// SIMATIC S7-200 SMART project (STEP 7-Micro/WIN SMART), CPU ST60

SYMBOL_TABLE V区符号
参数传输成功           V0.0     // 接收工控机传来的数据传输成功信号
参数是否更新           V0.1
挡板自动控制完成标志       V0.2
挡板电机开关           V0.3
挡板手动向内           V0.4
挡板手动向外           V0.5
挡板一键调节           V0.6
下料电机开关           V0.7
下料手动向前           V1.0
下料手动向后           V1.1
冷却电机开关           V1.2
冷却电机点动向内         V1.3
冷却电机点动向外         V1.4
冷柜一键调节           V1.5
调试按钮             V1.6
恢复出厂设置           V1.7
报警信息1用           VB2
V型架未处于停止位        V3.0     // 用于显示屏显示报警信息
系统处于急停模式         V3.1     // 用于显示屏显示报警信息
挡板运动超过左限制区       V3.2     // 用于显示屏显示报警信息
挡板运动超过右限制区       V3.3     // 用于显示屏显示报警信息
下料小车运动超过前限制      V3.4     // 用于显示屏显示报警信息
下料小车运动超过后限制      V3.5     // 用于显示屏显示报警信息
冷却风柜运动超过左限制      V3.6     // 用于显示屏显示报警信息
冷却风柜运动超过右限制      V3.7     // 用于显示屏显示报警信息
报警信息2用           VB4
上料步进故障           V5.0
上料传动故障           V5.1
上料夹料位报警          V5.2
请先建立绝对坐标         V5.3
链传动限位传感器报警       V5.4
挡板参数改变请初始化       V5.5
冷却参数改变请初始化       V5.6
报警灯红灯常开          V8.0
报警灯黄灯常开          V8.1
报警灯绿灯常开          V8.2
报警灯红灯闪烁和蜂鸣       V8.4
报警灯黄灯闪烁          V8.5
报警灯绿灯闪烁          V8.6
挡板电机手动运行         V10.0
冷却电机手动运行         V10.1
下料电机手动运行         V10.2
挡板手动一键调节         V10.3
挡板一键调节完成标志       V10.4
冷却手动一键调节         V10.5
冷却一键调节完成标志       V10.6
挡板点动向外           V11.1
挡板点动向内           V11.2
挡板电机查找原点按钮       V11.3
下料电机查找原点按钮       V11.4
冷却电机查找原点按钮       V11.5
挡板自动控制           V11.6
下料下移一个工位         V11.7
下料启动按钮           V12.0
下料手动完成标志         V12.1
下料手动回到原点         V12.2
下料手动回到底部         V12.3
冷却自动控制           V12.4
挡板电机查找原点         V12.5
下料电机查找原点         V12.6
冷却电机查找原点         V12.7
冷却点动向内           V13.0
冷却点动向外           V13.1
下料点动向前           V13.2
下料点动向后           V13.3
冷却启动按钮           V13.4
放料完成开关           V13.5    // 不再需要上杆件后，按下此按键，上料架上杆件自动向前
上料步进停止位          V13.6
上料杆件序号确认         V13.7
挡板电机CTRL错误参数     VB16
挡板电机RSEEK错误参数    VB18
挡板电机函数完成标志位      V20.1
挡板电机当前运动方向       V20.2
挡板电机查找原点完成位      V20.3    // 查找到原点动作已完成
挡板电机GOTO完成位      V20.4
挡板电机GOTO错误参数     VB21
挡板电机当前位置         VD24
挡板电机当前速度         VD28
上一次挡板停止位置        VD32
挡板电机移动位置         VD44
挡板电机速度           VD48
挡板电机移动模式         VB41
挡板电机停止运动轴        V40.1
挡板电机运动方向         V40.2
挡板当前实际位置         VD52
挡板相对运动距离         VD56
冷却电机初始化完成位       V60.1
冷却电机当前运动方向       V60.2
冷却电机查找原点完成位      V60.3
冷却电机GOTO完成位      V60.4
冷却电机GOTO错误参数     VB61
冷却电机当前位置         VD64
冷却电机当前速度         VD68
冷柜电机CTRL错误参数     VB72
冷柜电机RSEEK错误参数    VB75
冷却电机移动位置         VD84
冷却电机速度           VD88
冷却电机移动模式         VB81
冷却电机停止运动轴        V80.1
冷却电机运动方向         V80.2
下料电机函数完成标志位      V100.1
下料电机当前运动方向       V100.2
下料电机查找原点完成位      V100.3
下料电机GOTO完成位      V100.4
下料电机错误参数         VB101
下料电机当前位置         VD104
下料电机当前速度         VD108
下料电机当前位置上限       VD112
下料电机当前位置下限       VD116
下料电机移动位置         VD124
下料电机速度           VD128
下料电机移动模式         VB121
下料电机停止运动轴        V120.1
下料电机运动方向         V120.2
杆件编号             VB136
上一杆件数据           VD140
当前杆件数据           VD144
下料电机运动到杆件放置      VD150
下料电机下移一个杆件位      VD154
下料电机二号杆件位置       VD158
下料电机三号杆件位置       VD162
下料电机四号杆件位置       VD166
下料电机五号杆件位置       VD170
小车下料终点位置         VD174
挡板长度             VD180    // 定位零点以后，挡板能调节的最大长度
挡板预留长度           VD184    // 根据杆件的长度加上预留长度为实际调节距离
挡板临时变量           VD188    // 挡板长度减去当前杆件长度
挡板预留长度临时变量       VD192
轴0运动组态用          VB200    // VB200-VB292为轴0占用
轴1运动组态用          VB293    // VB293-VB385为轴1占用
轴2运动组态用          VB386    // VB386-VB478为轴2占用
链传动使能按钮          V480.0
链传动低速按钮          V480.1
链传动高速按钮          V480.2
链传动一个工位按钮        V480.3   // 链传动机构运动一个杆位按钮
链传动自动运行          V480.4
杆件编号1            V500.0   // VB500-VB748存放杆件编号和长度
杆件编号2            V500.1   // VB500-VB748存放杆件编号和长度
杆件编号3            V500.2   // VB500-VB748存放杆件编号和长度
杆件编号4            V500.3   // VB500-VB748存放杆件编号和长度
杆件编号5            V500.4   // VB500-VB748存放杆件编号和长度
杆件编号6            V500.5   // VB500-VB748存放杆件编号和长度
杆件编号7            V500.6   // VB500-VB748存放杆件编号和长度
杆件编号8            V500.7   // VB500-VB748存放杆件编号和长度
杆件编号9            V501.0   // VB500-VB748存放杆件编号和长度
杆件编号10           V501.1   // VB500-VB748存放杆件编号和长度
杆件编号11           V501.2   // VB500-VB748存放杆件编号和长度
杆件编号12           V501.3   // VB500-VB748存放杆件编号和长度
杆件编号13           V501.4   // VB500-VB748存放杆件编号和长度
杆件编号14           V501.5   // VB500-VB748存放杆件编号和长度
杆件编号15           V501.6   // VB500-VB748存放杆件编号和长度
杆件编号16           V501.7   // VB500-VB748存放杆件编号和长度
杆件编号17           V502.0   // VB500-VB748存放杆件编号和长度
杆件编号18           V502.1   // VB500-VB748存放杆件编号和长度
杆件编号19           V502.2   // VB500-VB748存放杆件编号和长度
杆件编号20           V502.3   // VB500-VB748存放杆件编号和长度
杆件编号21           V502.4   // VB500-VB748存放杆件编号和长度
杆件编号22           V502.5   // VB500-VB748存放杆件编号和长度
杆件编号23           V502.6   // VB500-VB748存放杆件编号和长度
杆件编号24           V502.7   // VB500-VB748存放杆件编号和长度
杆件编号25           V503.0   // VB500-VB748存放杆件编号和长度
杆件编号26           V503.1   // VB500-VB748存放杆件编号和长度
杆件编号27           V503.2   // VB500-VB748存放杆件编号和长度
杆件编号28           V503.3   // VB500-VB748存放杆件编号和长度
杆件编号29           V503.4   // VB500-VB748存放杆件编号和长度
杆件编号30           V503.5   // VB500-VB748存放杆件编号和长度
杆件编号31           V503.6   // VB500-VB748存放杆件编号和长度
杆件编号32           V503.7   // VB500-VB748存放杆件编号和长度
杆件编号33           V504.0   // VB500-VB748存放杆件编号和长度
杆件编号34           V504.1   // VB500-VB748存放杆件编号和长度
杆件编号35           V504.2   // VB500-VB748存放杆件编号和长度
杆件编号36           V504.3   // VB500-VB748存放杆件编号和长度
杆件编号37           V504.4   // VB500-VB748存放杆件编号和长度
杆件编号38           V504.5   // VB500-VB748存放杆件编号和长度
杆件编号39           V504.6   // VB500-VB748存放杆件编号和长度
杆件编号40           V504.7   // VB500-VB748存放杆件编号和长度
杆件编号41           V505.0   // VB500-VB748存放杆件编号和长度
杆件编号42           V505.1   // VB500-VB748存放杆件编号和长度
杆件编号43           V505.2   // VB500-VB748存放杆件编号和长度
杆件编号44           V505.3   // VB500-VB748存放杆件编号和长度
杆件编号45           V505.4   // VB500-VB748存放杆件编号和长度
杆件编号46           V505.5   // VB500-VB748存放杆件编号和长度
杆件编号47           V505.6   // VB500-VB748存放杆件编号和长度
杆件编号48           V505.7   // VB500-VB748存放杆件编号和长度
杆件编号49           V506.0   // VB500-VB748存放杆件编号和长度
杆件编号50           V506.1   // VB500-VB748存放杆件编号和长度
杆件编号临时变量         VB510
杆件编号标志位1         V520.1
杆件编号标志位2         V520.2
杆件编号标志位3         V520.3
杆件编号标志位4         V520.4
杆件编号标志位5         V520.5
杆件编号标志位6         V520.6
杆件编号标志位7         V520.7
杆件编号标志位8         V521.0
杆件编号标志位9         V521.1
杆件编号标志位10        V521.2
杆件编号标志位11        V521.3
杆件编号标志位12        V521.4
杆件编号标志位13        V521.5
杆件编号标志位14        V521.6
杆件编号标志位15        V521.7
杆件编号标志位16        V522.0
杆件编号标志位17        V522.1
杆件编号标志位18        V522.2
杆件编号标志位19        V522.3
杆件编号标志位20        V522.4
杆件编号标志位21        V522.5
杆件编号标志位22        V522.6
杆件编号标志位23        V522.7
杆件编号标志位24        V523.0
杆件编号标志位25        V523.1
杆件编号标志位26        V523.2
杆件编号标志位27        V523.3
杆件编号标志位28        V523.4
杆件编号标志位29        V523.5
杆件编号标志位30        V523.6
杆件编号标志位31        V523.7
杆件编号标志位32        V524.0
杆件编号标志位33        V524.1
杆件编号标志位34        V524.2
杆件编号标志位35        V524.3
杆件编号标志位36        V524.4
杆件编号标志位37        V524.5
杆件编号标志位38        V524.6
杆件编号标志位39        V524.7
杆件编号标志位40        V525.0
杆件编号标志位41        V525.1
杆件编号标志位42        V525.2
杆件编号标志位43        V525.3
杆件编号标志位44        V525.4
杆件编号标志位45        V525.5
杆件编号标志位46        V525.6
杆件编号标志位47        V525.7
杆件编号标志位48        V526.0
杆件编号标志位49        V526.1
杆件编号标志位50        V526.2
上料架位置1           VB540
上料架位置2           VB541
上料架位置3           VB542
上料架位置4           VB543
上料架位置5           VB544
上料架位置6           VB545
上料架位置7           VB546
上料架位置8           VB547
上料架位置9           VB548
上料架位置10          VB549
上料架位置11          VB550
上料架位置12          VB551
上料架位置13          VB552
上料架位置14          VB553
上料架位置15          VB554
上料架位置16          VB555
上料架位置17          VB556
上料架位置18          VB557
上料架位置19          VB558
上料架位置20          VB559
上料架位置21          VB560
上料架位置22          VB561
上料架位置23          VB562
上料架位置24          VB563
上料架位置25          VB564
上料架位置26          VB565
上料架位置27          VB566
上料架位置28          VB567
上料架位置29          VB568
上料架位置30          VB569
上料架位置31          VB570
上料架位置32          VB571
上料架标志位1          V580.0
上料架标志位2          V580.1
上料架标志位3          V580.2
顺序控制延时1          VW800    // T33定时变量
顺序控制延时2          VW802    // T34定时变量
挡板手动调节延时         VW804    // T104定时变量
上料故障报警定时         VW806    // T37定时变量
链传动控制定时器         VW808    // T97定时变量
挡板运动脉冲1          VW810    // T101定时变量
下料运动脉冲1          VW812    // T102定时变量
冷却运动脉冲1          VW814    // T103定时变量
上料停止位判断定时器       VW816    // T34定时变量
冷却手动调节延时         VW818    // T105定时变量
冷柜长度             VD900    // 定位零点以后，冷却风扇能移动的最大长度
冷柜预留长度           VD904    // 冷柜长度减去杆的长度
冷柜临时变量           VD908
冷柜预留长度临时变量       VD912
挡调距离             VD916
柜调长度             VD920
下料电机当前位置temp     VD924
下料运动左区间          VD928
下料运动右区间          VD932
下料电机速度高速         VD936    // 下料变速运动，速度为高速
下料电机速度低速         VD940    // 下料变速运动，速度为低速
前后两根杆件长度差        VD960
冷柜上一杆件长度         VD964
冷柜当前杆件长度         VD968
冷柜前后杆件长度差        VD972
风柜当前实际位置         VD976
上一次风柜停止位置        VD980
风柜相对移动距离         VD984
置工件就绪            V1000.0
上料位异常信号          V1001.0
下料位允许放料信号        V1018.0
下料位启动信号          V1118.1
下料位异常信号          V1019.0
上料取件完成信号         V1200.0
下料位机器人放料完成信      V1212.0
下料小车下移信号         V1212.1
手动机器人放料完成信号      V1212.2
temp上料位异常信号      V1500.0
temp下料位异常信号      V1500.1
temp冷却位异常信号      V1500.2
挡板电机手动完成标志       VB1600
冷却电机手动完成标志       VB1602
手动跳到s_6          V3000.0
C0计数器复位          V5000.0
END_SYMBOL_TABLE

SYMBOL_TABLE 系统符号
Always_On        SM0.0    // 始终接通
First_Scan_On    SM0.1    // 仅在第一个扫描周期时接通
END_SYMBOL_TABLE

SYMBOL_TABLE S区符号
扫码启动上料           S0.0
判断杆件长度是否更新       S0.1
挡板调节             S0.2
判断夹料位是否有杆件       S0.3
开启链传动            S0.4
停止链传动            S0.5
置工件就绪回到第一步       S0.6
END_SYMBOL_TABLE

SYMBOL_TABLE 定时器符号
顺序控制延时1_10ms     T33      // 短延时，保证正确读取到判断工件有无传感器的状态
上料停止位判断延时_10ms   T34
到位传感器延时_10ms     T35      // 短延时，保证正确读取到判断工件有无传感器的状态
顺序控制延时3_100ms    T36
上料故障报警定时_100ms   T37      // 设置定时，超时则报警
下料减速区脉冲_100ms    T39
上料初始化调试          T38
链传动控制定时器_10ms    T97      // 确保链传动走出当前传感器感应区，能接收到下一个传感器信号
挡板运动脉冲1_100ms    T101     // 给一个运动脉冲信号，挡板移动到杆件长度处
下料运动脉冲1_100ms    T102     // 给一个运动脉冲信号，小车移动到机器人放料处
冷却运动脉冲1_100ms    T103     // 给一个运动脉冲信号，风柜移动到杆件长度处
挡板手动调节延时_100ms   T104     // 手动调节结束后，延时一定时间，待电机当前位置稳定后再读取
冷却手动调节街延时_100m   T105     // 手动调节结束后，延时一定时间，待电机当前位置稳定后再读取
报警灯红灯高电平_100ms   T120
报警灯红灯低电平_100ms   T121
报警灯黄灯高电平_100ms   T122
报警灯黄灯低电平_100ms   T123
报警灯绿灯高电平_100ms   T124
报警灯绿灯低电平_100ms   T125
报警蜂鸣器高电平_100ms   T126
报警蜂鸣器低电平_100ms   T127
END_SYMBOL_TABLE

ORGANIZATION_BLOCK 主程序:OB1
TITLE=
BEGIN
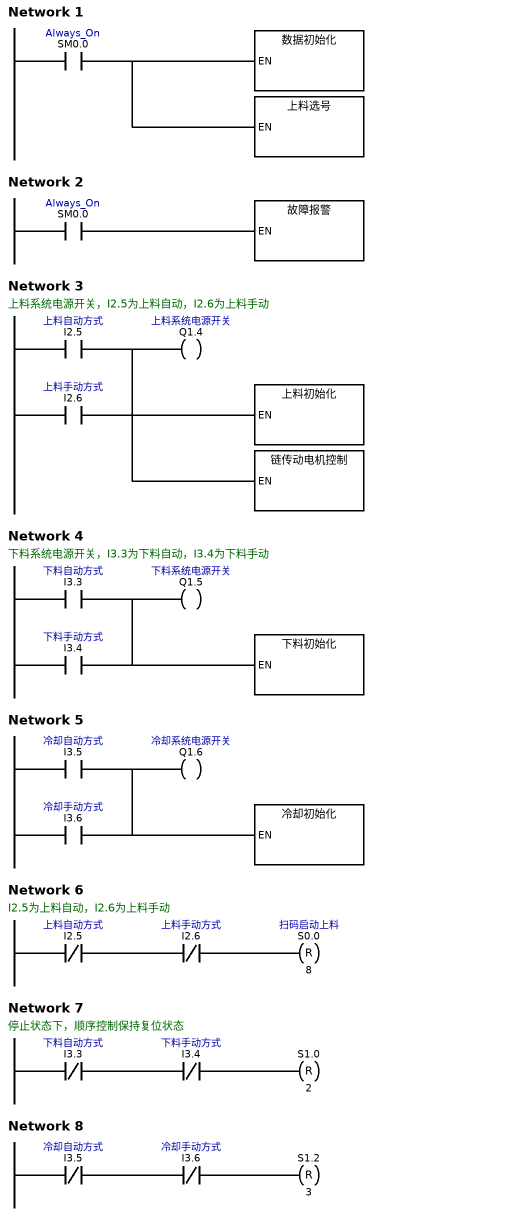
Network 1
LD     Always_On:SM0.0
CALL   数据初始化:SBR20
CALL   上料选号:SBR17
Network 2
LD     Always_On:SM0.0
CALL   故障报警:SBR21
Network 3
// 上料系统电源开关，I2.5为上料自动，I2.6为上料手动
LD     上料自动方式:I2.5
O      上料手动方式:I2.6
=      上料系统电源开关:Q1.4
CALL   上料初始化:SBR14
CALL   链传动电机控制:SBR19
Network 4
// 下料系统电源开关，I3.3为下料自动，I3.4为下料手动
LD     下料自动方式:I3.3
O      下料手动方式:I3.4
=      下料系统电源开关:Q1.5
CALL   下料初始化:SBR15
Network 5
LD     冷却自动方式:I3.5
O      冷却手动方式:I3.6
=      冷却系统电源开关:Q1.6
CALL   冷却初始化:SBR16
Network 6
// I2.5为上料自动，I2.6为上料手动
LDN    上料自动方式:I2.5
AN     上料手动方式:I2.6
R      扫码启动上料:S0.0, 8
Network 7
// 停止状态下，顺序控制保持复位状态
LDN    下料自动方式:I3.3
AN     下料手动方式:I3.4
R      S1.0, 2
Network 8
LDN    冷却自动方式:I3.5
AN     冷却手动方式:I3.6
R      S1.2, 3
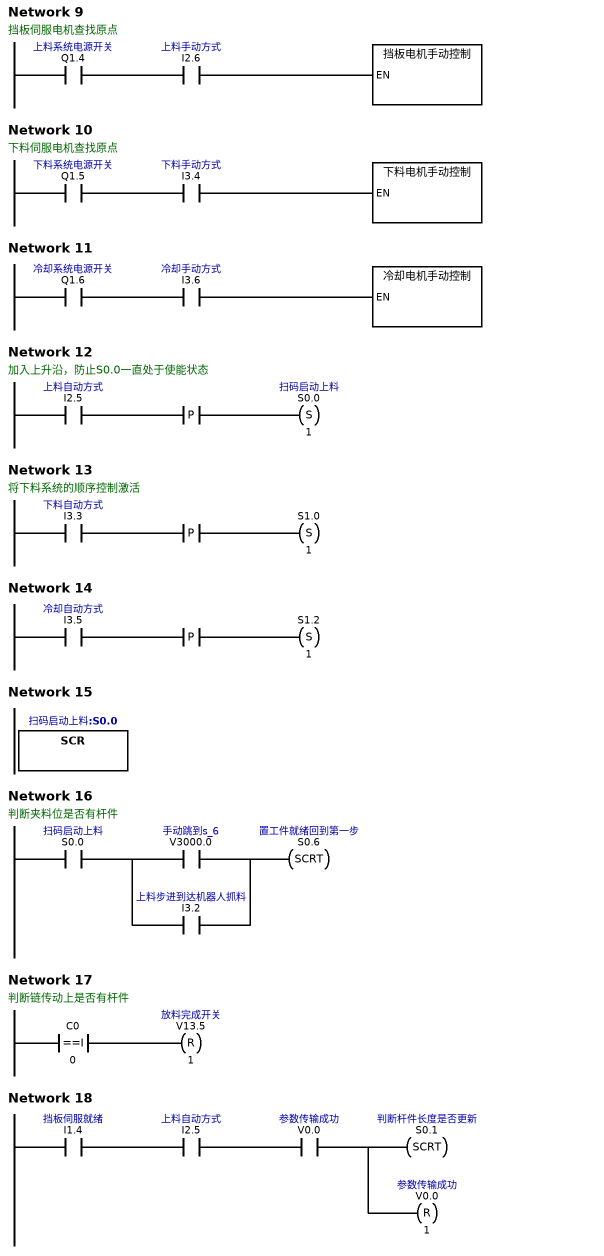
Network 9
// 挡板伺服电机查找原点
LD     上料系统电源开关:Q1.4
A      上料手动方式:I2.6
CALL   挡板电机手动控制:SBR7
Network 10
// 下料伺服电机查找原点
LD     下料系统电源开关:Q1.5
A      下料手动方式:I3.4
CALL   下料电机手动控制:SBR9
Network 11
LD     冷却系统电源开关:Q1.6
A      冷却手动方式:I3.6
CALL   冷却电机手动控制:SBR18
Network 12
// 加入上升沿，防止S0.0一直处于使能状态
LD     上料自动方式:I2.5
EU
S      扫码启动上料:S0.0, 1
Network 13
// 将下料系统的顺序控制激活
LD     下料自动方式:I3.3
EU
S      S1.0, 1
Network 14
LD     冷却自动方式:I3.5
EU
S      S1.2, 1
Network 15
LSCR   扫码启动上料:S0.0
Network 16
// 判断夹料位是否有杆件
LD     扫码启动上料:S0.0
LD     手动跳到s_6:V3000.0
O      上料步进到达机器人抓料:I3.2
ALD
SCRT   置工件就绪回到第一步:S0.6
Network 17
// 判断链传动上是否有杆件
LDW=   C0, 0
R      放料完成开关:V13.5, 1
Network 18
LD     挡板伺服就绪:I1.4
A      上料自动方式:I2.5
A      参数传输成功:V0.0
SCRT   判断杆件长度是否更新:S0.1
R      参数传输成功:V0.0, 1
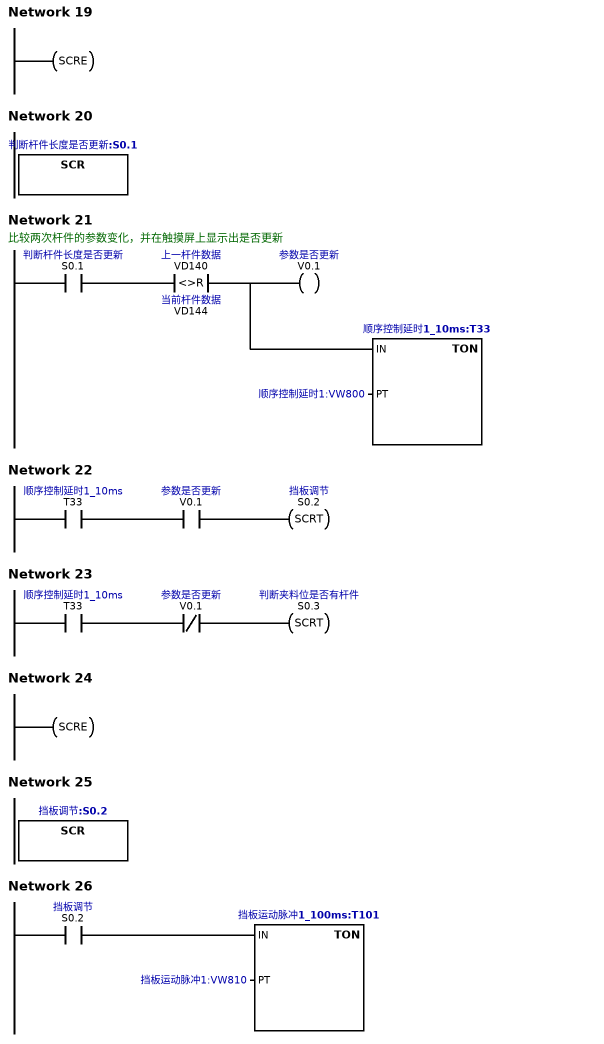
Network 19
SCRE
Network 20
LSCR   判断杆件长度是否更新:S0.1
Network 21
// 比较两次杆件的参数变化，并在触摸屏上显示出是否更新
LD     判断杆件长度是否更新:S0.1
AR<>   上一杆件数据:VD140, 当前杆件数据:VD144
=      参数是否更新:V0.1
TON    顺序控制延时1_10ms:T33, 顺序控制延时1:VW800
Network 22
LD     顺序控制延时1_10ms:T33
A      参数是否更新:V0.1
SCRT   挡板调节:S0.2
Network 23
LD     顺序控制延时1_10ms:T33
AN     参数是否更新:V0.1
SCRT   判断夹料位是否有杆件:S0.3
Network 24
SCRE
Network 25
LSCR   挡板调节:S0.2
Network 26
LD     挡板调节:S0.2
TON    挡板运动脉冲1_100ms:T101, 挡板运动脉冲1:VW810
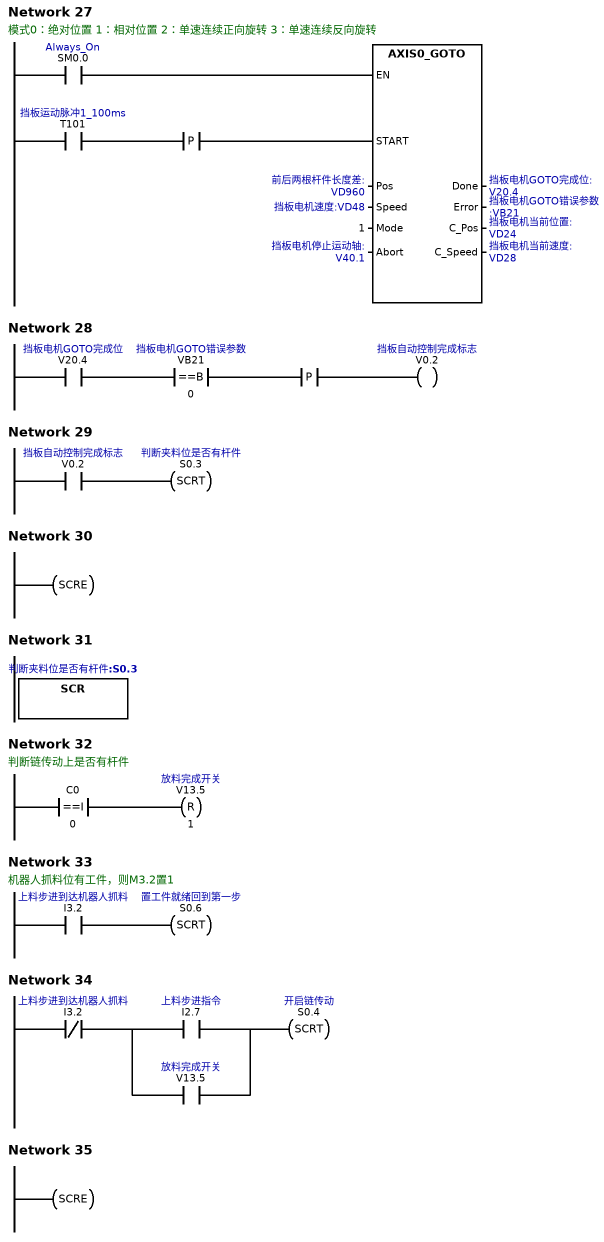
Network 27
// 模式0：绝对位置 1：相对位置 2：单速连续正向旋转 3：单速连续反向旋转
LD     Always_On:SM0.0
=      L60.0
LD     挡板运动脉冲1_100ms:T101
EU
=      L63.7
LD     L60.0
CALL   AXIS0_GOTO:SBR2, L63.7, 前后两根杆件长度差:VD960, 挡板电机速度:VD48, 1, 挡板电机停止运动轴:V40.1, 挡板电机GOTO完成位:V20.4, 挡板电机GOTO错误参数:VB21, 挡板电机当前位置:VD24, 挡板电机当前速度:VD28
Network 28
LD     挡板电机GOTO完成位:V20.4
AB=    挡板电机GOTO错误参数:VB21, 0
EU
=      挡板自动控制完成标志:V0.2
Network 29
LD     挡板自动控制完成标志:V0.2
SCRT   判断夹料位是否有杆件:S0.3
Network 30
SCRE
Network 31
LSCR   判断夹料位是否有杆件:S0.3
Network 32
// 判断链传动上是否有杆件
LDW=   C0, 0
R      放料完成开关:V13.5, 1
Network 33
// 机器人抓料位有工件，则M3.2置1
LD     上料步进到达机器人抓料:I3.2
SCRT   置工件就绪回到第一步:S0.6
Network 34
LDN    上料步进到达机器人抓料:I3.2
LD     上料步进指令:I2.7
O      放料完成开关:V13.5
ALD
SCRT   开启链传动:S0.4
Network 35
SCRE
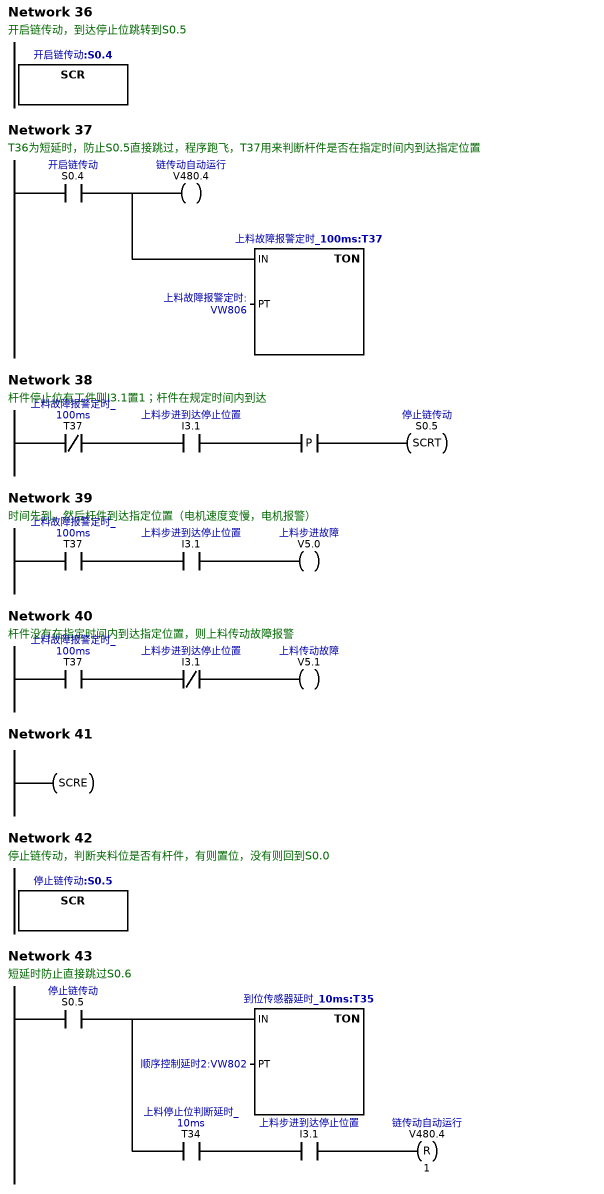
Network 36
// 开启链传动，到达停止位跳转到S0.5
LSCR   开启链传动:S0.4
Network 37
// T36为短延时，防止S0.5直接跳过，程序跑飞，T37用来判断杆件是否在指定时间内到达指定位置
LD     开启链传动:S0.4
=      链传动自动运行:V480.4
TON    上料故障报警定时_100ms:T37, 上料故障报警定时:VW806
Network 38
// 杆件停止位有工件则I3.1置1；杆件在规定时间内到达
LDN    上料故障报警定时_100ms:T37
A      上料步进到达停止位置:I3.1
EU
SCRT   停止链传动:S0.5
Network 39
// 时间先到，然后杆件到达指定位置（电机速度变慢，电机报警）
LD     上料故障报警定时_100ms:T37
A      上料步进到达停止位置:I3.1
=      上料步进故障:V5.0
Network 40
// 杆件没有在指定时间内到达指定位置，则上料传动故障报警
LD     上料故障报警定时_100ms:T37
AN     上料步进到达停止位置:I3.1
=      上料传动故障:V5.1
Network 41
SCRE
Network 42
// 停止链传动，判断夹料位是否有杆件，有则置位，没有则回到S0.0
LSCR   停止链传动:S0.5
Network 43
// 短延时防止直接跳过S0.6
LD     停止链传动:S0.5
TON    到位传感器延时_10ms:T35, 顺序控制延时2:VW802
A      上料停止位判断延时_10ms:T34
A      上料步进到达停止位置:I3.1
R      链传动自动运行:V480.4, 1
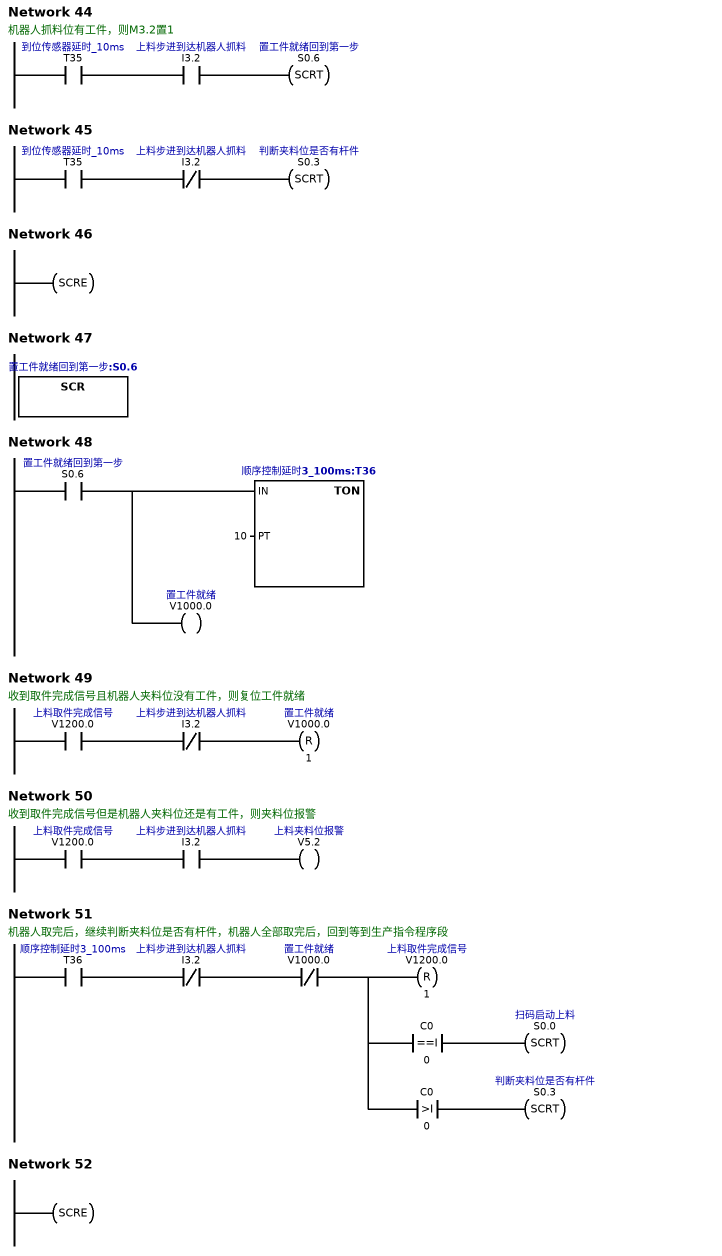
Network 44
// 机器人抓料位有工件，则M3.2置1
LD     到位传感器延时_10ms:T35
A      上料步进到达机器人抓料:I3.2
SCRT   置工件就绪回到第一步:S0.6
Network 45
LD     到位传感器延时_10ms:T35
AN     上料步进到达机器人抓料:I3.2
SCRT   判断夹料位是否有杆件:S0.3
Network 46
SCRE
Network 47
LSCR   置工件就绪回到第一步:S0.6
Network 48
LD     置工件就绪回到第一步:S0.6
TON    顺序控制延时3_100ms:T36, 10
=      置工件就绪:V1000.0
Network 49
// 收到取件完成信号且机器人夹料位没有工件，则复位工件就绪
LD     上料取件完成信号:V1200.0
AN     上料步进到达机器人抓料:I3.2
R      置工件就绪:V1000.0, 1
Network 50
// 收到取件完成信号但是机器人夹料位还是有工件，则夹料位报警
LD     上料取件完成信号:V1200.0
A      上料步进到达机器人抓料:I3.2
=      上料夹料位报警:V5.2
Network 51
// 机器人取完后，继续判断夹料位是否有杆件，机器人全部取完后，回到等到生产指令程序段
LD     顺序控制延时3_100ms:T36
AN     上料步进到达机器人抓料:I3.2
AN     置工件就绪:V1000.0
LPS
R      上料取件完成信号:V1200.0, 1
AW=    C0, 0
SCRT   扫码启动上料:S0.0
LPP
AW>    C0, 0
SCRT   判断夹料位是否有杆件:S0.3
Network 52
SCRE
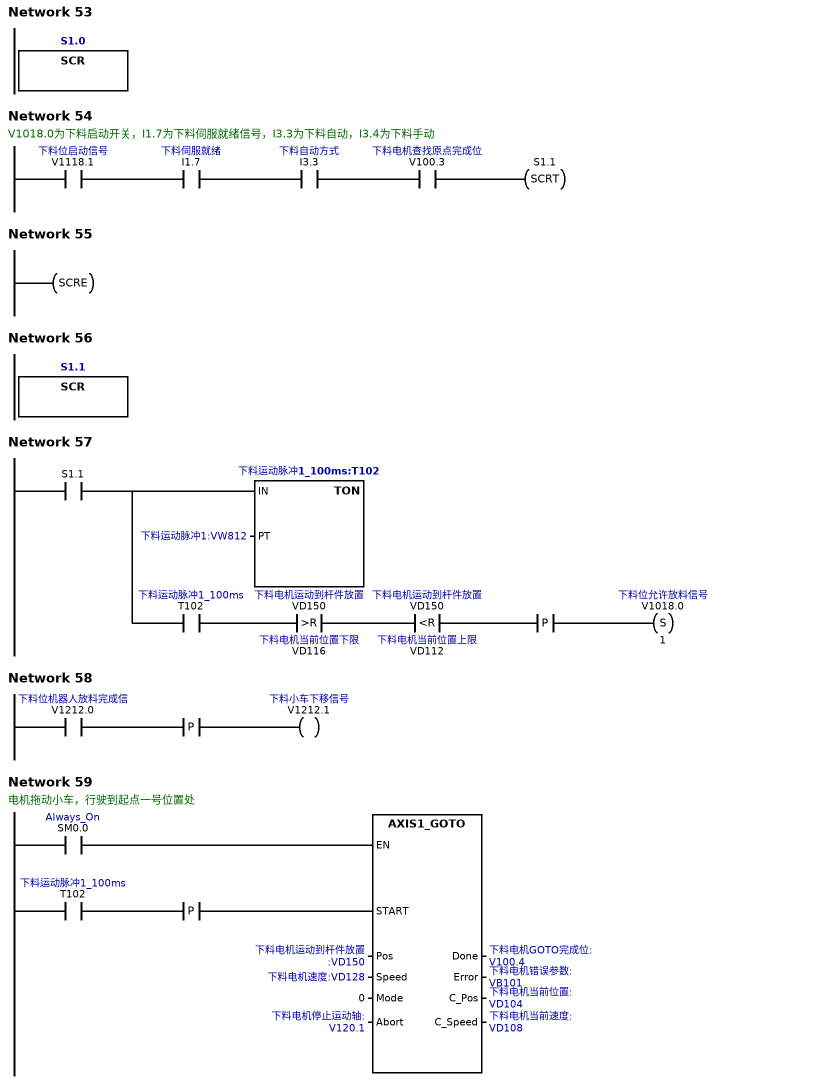
Network 53
LSCR   S1.0
Network 54
// V1018.0为下料启动开关，I1.7为下料伺服就绪信号，I3.3为下料自动，I3.4为下料手动
LD     下料位启动信号:V1118.1
A      下料伺服就绪:I1.7
A      下料自动方式:I3.3
A      下料电机查找原点完成位:V100.3
SCRT   S1.1
Network 55
SCRE
Network 56
LSCR   S1.1
Network 57
LD     S1.1
TON    下料运动脉冲1_100ms:T102, 下料运动脉冲1:VW812
A      下料运动脉冲1_100ms:T102
AR>    下料电机运动到杆件放置:VD150, 下料电机当前位置下限:VD116
AR<    下料电机运动到杆件放置:VD150, 下料电机当前位置上限:VD112
EU
S      下料位允许放料信号:V1018.0, 1
Network 58
LD     下料位机器人放料完成信:V1212.0
EU
=      下料小车下移信号:V1212.1
Network 59
// 电机拖动小车，行驶到起点一号位置处
LD     Always_On:SM0.0
=      L60.0
LD     下料运动脉冲1_100ms:T102
EU
=      L63.7
LD     L60.0
CALL   AXIS1_GOTO:SBR6, L63.7, 下料电机运动到杆件放置:VD150, 下料电机速度:VD128, 0, 下料电机停止运动轴:V120.1, 下料电机GOTO完成位:V100.4, 下料电机错误参数:VB101, 下料电机当前位置:VD104, 下料电机当前速度:VD108
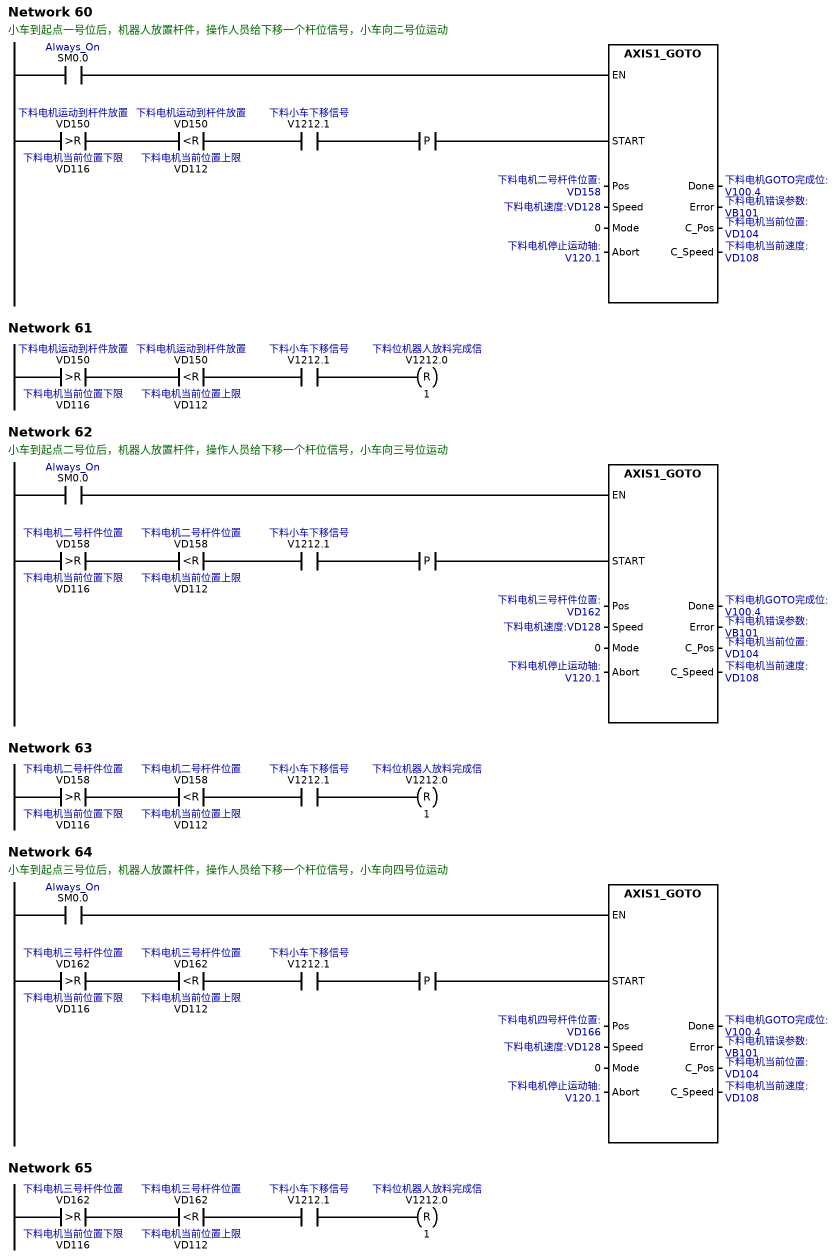
Network 60
// 小车到起点一号位后，机器人放置杆件，操作人员给下移一个杆位信号，小车向二号位运动
LD     Always_On:SM0.0
=      L60.0
LDR>   下料电机运动到杆件放置:VD150, 下料电机当前位置下限:VD116
AR<    下料电机运动到杆件放置:VD150, 下料电机当前位置上限:VD112
A      下料小车下移信号:V1212.1
EU
=      L63.7
LD     L60.0
CALL   AXIS1_GOTO:SBR6, L63.7, 下料电机二号杆件位置:VD158, 下料电机速度:VD128, 0, 下料电机停止运动轴:V120.1, 下料电机GOTO完成位:V100.4, 下料电机错误参数:VB101, 下料电机当前位置:VD104, 下料电机当前速度:VD108
Network 61
LDR>   下料电机运动到杆件放置:VD150, 下料电机当前位置下限:VD116
AR<    下料电机运动到杆件放置:VD150, 下料电机当前位置上限:VD112
A      下料小车下移信号:V1212.1
R      下料位机器人放料完成信:V1212.0, 1
Network 62
// 小车到起点二号位后，机器人放置杆件，操作人员给下移一个杆位信号，小车向三号位运动
LD     Always_On:SM0.0
=      L60.0
LDR>   下料电机二号杆件位置:VD158, 下料电机当前位置下限:VD116
AR<    下料电机二号杆件位置:VD158, 下料电机当前位置上限:VD112
A      下料小车下移信号:V1212.1
EU
=      L63.7
LD     L60.0
CALL   AXIS1_GOTO:SBR6, L63.7, 下料电机三号杆件位置:VD162, 下料电机速度:VD128, 0, 下料电机停止运动轴:V120.1, 下料电机GOTO完成位:V100.4, 下料电机错误参数:VB101, 下料电机当前位置:VD104, 下料电机当前速度:VD108
Network 63
LDR>   下料电机二号杆件位置:VD158, 下料电机当前位置下限:VD116
AR<    下料电机二号杆件位置:VD158, 下料电机当前位置上限:VD112
A      下料小车下移信号:V1212.1
R      下料位机器人放料完成信:V1212.0, 1
Network 64
// 小车到起点三号位后，机器人放置杆件，操作人员给下移一个杆位信号，小车向四号位运动
LD     Always_On:SM0.0
=      L60.0
LDR>   下料电机三号杆件位置:VD162, 下料电机当前位置下限:VD116
AR<    下料电机三号杆件位置:VD162, 下料电机当前位置上限:VD112
A      下料小车下移信号:V1212.1
EU
=      L63.7
LD     L60.0
CALL   AXIS1_GOTO:SBR6, L63.7, 下料电机四号杆件位置:VD166, 下料电机速度:VD128, 0, 下料电机停止运动轴:V120.1, 下料电机GOTO完成位:V100.4, 下料电机错误参数:VB101, 下料电机当前位置:VD104, 下料电机当前速度:VD108
Network 65
LDR>   下料电机三号杆件位置:VD162, 下料电机当前位置下限:VD116
AR<    下料电机三号杆件位置:VD162, 下料电机当前位置上限:VD112
A      下料小车下移信号:V1212.1
R      下料位机器人放料完成信:V1212.0, 1
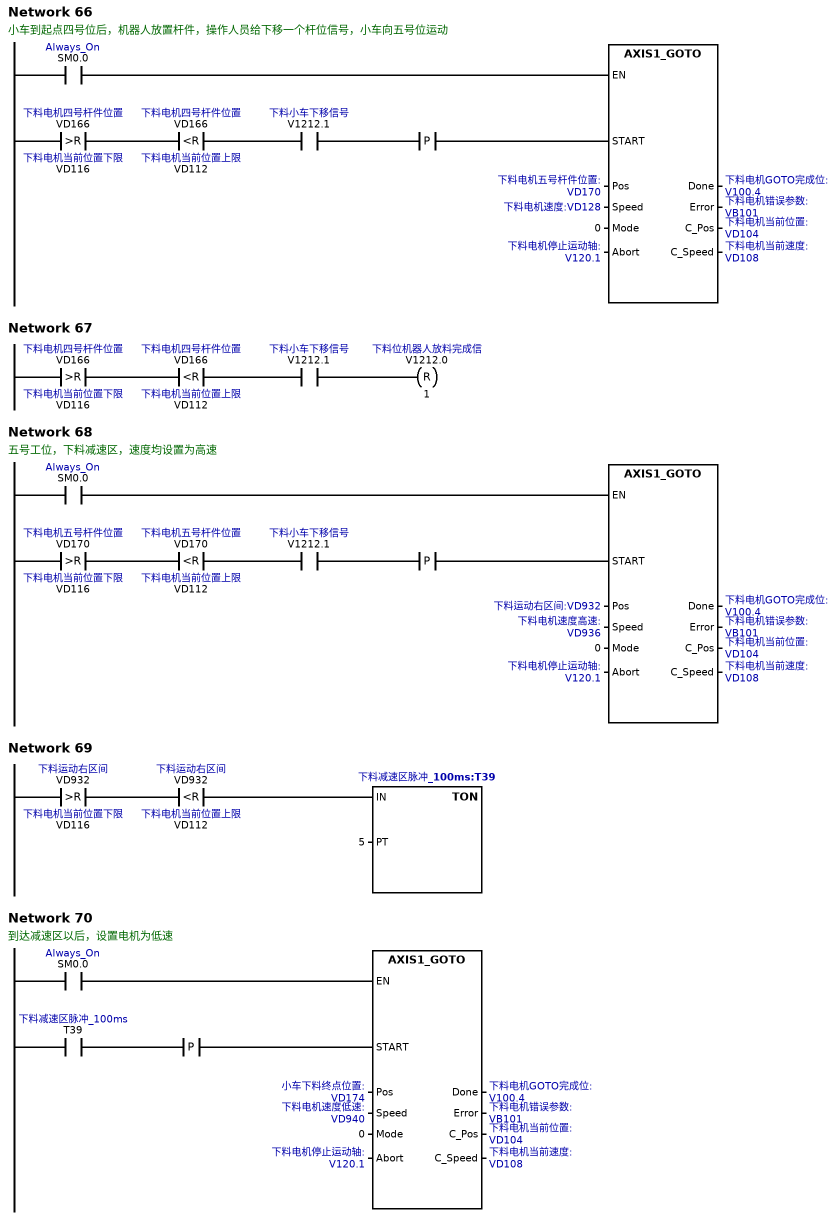
Network 66
// 小车到起点四号位后，机器人放置杆件，操作人员给下移一个杆位信号，小车向五号位运动
LD     Always_On:SM0.0
=      L60.0
LDR>   下料电机四号杆件位置:VD166, 下料电机当前位置下限:VD116
AR<    下料电机四号杆件位置:VD166, 下料电机当前位置上限:VD112
A      下料小车下移信号:V1212.1
EU
=      L63.7
LD     L60.0
CALL   AXIS1_GOTO:SBR6, L63.7, 下料电机五号杆件位置:VD170, 下料电机速度:VD128, 0, 下料电机停止运动轴:V120.1, 下料电机GOTO完成位:V100.4, 下料电机错误参数:VB101, 下料电机当前位置:VD104, 下料电机当前速度:VD108
Network 67
LDR>   下料电机四号杆件位置:VD166, 下料电机当前位置下限:VD116
AR<    下料电机四号杆件位置:VD166, 下料电机当前位置上限:VD112
A      下料小车下移信号:V1212.1
R      下料位机器人放料完成信:V1212.0, 1
Network 68
// 五号工位，下料减速区，速度均设置为高速
LD     Always_On:SM0.0
=      L60.0
LDR>   下料电机五号杆件位置:VD170, 下料电机当前位置下限:VD116
AR<    下料电机五号杆件位置:VD170, 下料电机当前位置上限:VD112
A      下料小车下移信号:V1212.1
EU
=      L63.7
LD     L60.0
CALL   AXIS1_GOTO:SBR6, L63.7, 下料运动右区间:VD932, 下料电机速度高速:VD936, 0, 下料电机停止运动轴:V120.1, 下料电机GOTO完成位:V100.4, 下料电机错误参数:VB101, 下料电机当前位置:VD104, 下料电机当前速度:VD108
Network 69
LDR>   下料运动右区间:VD932, 下料电机当前位置下限:VD116
AR<    下料运动右区间:VD932, 下料电机当前位置上限:VD112
TON    下料减速区脉冲_100ms:T39, 5
Network 70
// 到达减速区以后，设置电机为低速
LD     Always_On:SM0.0
=      L60.0
LD     下料减速区脉冲_100ms:T39
EU
=      L63.7
LD     L60.0
CALL   AXIS1_GOTO:SBR6, L63.7, 小车下料终点位置:VD174, 下料电机速度低速:VD940, 0, 下料电机停止运动轴:V120.1, 下料电机GOTO完成位:V100.4, 下料电机错误参数:VB101, 下料电机当前位置:VD104, 下料电机当前速度:VD108
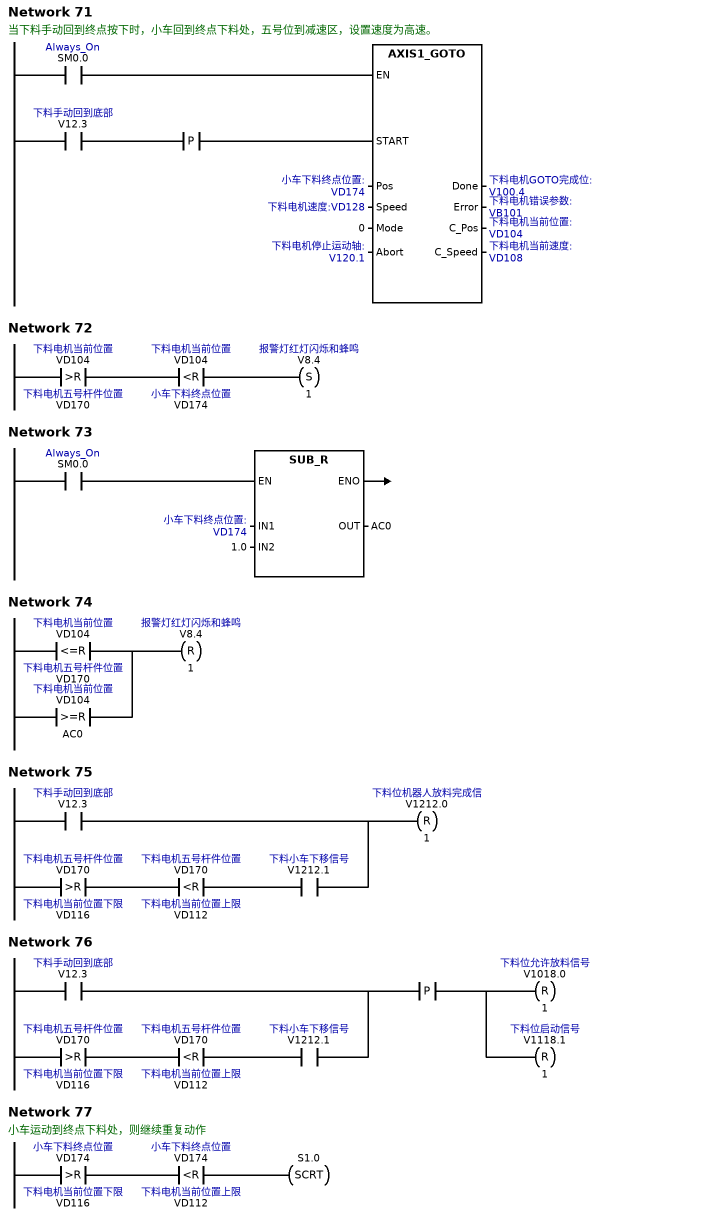
Network 71
// 当下料手动回到终点按下时，小车回到终点下料处，五号位到减速区，设置速度为高速。
LD     Always_On:SM0.0
=      L60.0
LD     下料手动回到底部:V12.3
EU
=      L63.7
LD     L60.0
CALL   AXIS1_GOTO:SBR6, L63.7, 小车下料终点位置:VD174, 下料电机速度:VD128, 0, 下料电机停止运动轴:V120.1, 下料电机GOTO完成位:V100.4, 下料电机错误参数:VB101, 下料电机当前位置:VD104, 下料电机当前速度:VD108
Network 72
LDR>   下料电机当前位置:VD104, 下料电机五号杆件位置:VD170
AR<    下料电机当前位置:VD104, 小车下料终点位置:VD174
S      报警灯红灯闪烁和蜂鸣:V8.4, 1
Network 73
LD     Always_On:SM0.0
MOVR   小车下料终点位置:VD174, AC0
-R     1.0, AC0
Network 74
LDR<=  下料电机当前位置:VD104, 下料电机五号杆件位置:VD170
OR>=   下料电机当前位置:VD104, AC0
R      报警灯红灯闪烁和蜂鸣:V8.4, 1
Network 75
LD     下料手动回到底部:V12.3
LDR>   下料电机五号杆件位置:VD170, 下料电机当前位置下限:VD116
AR<    下料电机五号杆件位置:VD170, 下料电机当前位置上限:VD112
A      下料小车下移信号:V1212.1
OLD
R      下料位机器人放料完成信:V1212.0, 1
Network 76
LD     下料手动回到底部:V12.3
LDR>   下料电机五号杆件位置:VD170, 下料电机当前位置下限:VD116
AR<    下料电机五号杆件位置:VD170, 下料电机当前位置上限:VD112
A      下料小车下移信号:V1212.1
OLD
EU
R      下料位允许放料信号:V1018.0, 1
R      下料位启动信号:V1118.1, 1
Network 77
// 小车运动到终点下料处，则继续重复动作
LDR>   小车下料终点位置:VD174, 下料电机当前位置下限:VD116
AR<    小车下料终点位置:VD174, 下料电机当前位置上限:VD112
SCRT   S1.0
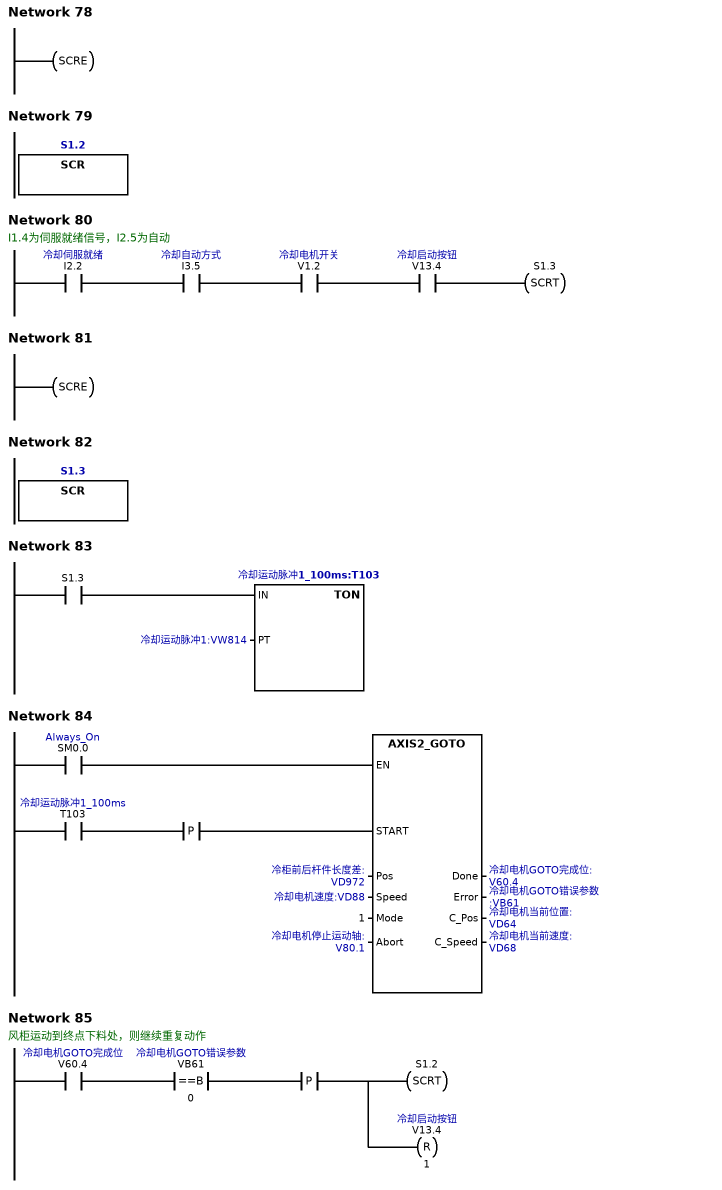
Network 78
SCRE
Network 79
LSCR   S1.2
Network 80
// I1.4为伺服就绪信号，I2.5为自动
LD     冷却伺服就绪:I2.2
A      冷却自动方式:I3.5
A      冷却电机开关:V1.2
A      冷却启动按钮:V13.4
SCRT   S1.3
Network 81
SCRE
Network 82
LSCR   S1.3
Network 83
LD     S1.3
TON    冷却运动脉冲1_100ms:T103, 冷却运动脉冲1:VW814
Network 84
LD     Always_On:SM0.0
=      L60.0
LD     冷却运动脉冲1_100ms:T103
EU
=      L63.7
LD     L60.0
CALL   AXIS2_GOTO:SBR12, L63.7, 冷柜前后杆件长度差:VD972, 冷却电机速度:VD88, 1, 冷却电机停止运动轴:V80.1, 冷却电机GOTO完成位:V60.4, 冷却电机GOTO错误参数:VB61, 冷却电机当前位置:VD64, 冷却电机当前速度:VD68
Network 85
// 风柜运动到终点下料处，则继续重复动作
LD     冷却电机GOTO完成位:V60.4
AB=    冷却电机GOTO错误参数:VB61, 0
EU
SCRT   S1.2
R      冷却启动按钮:V13.4, 1
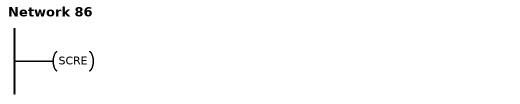
Network 86
SCRE
END_ORGANIZATION_BLOCK

// SBR0: protected block, not included

// SBR1: protected block, not included

// SBR2: protected block, not included

// SBR3: protected block, not included

// SBR4: protected block, not included

// SBR5: protected block, not included

// SBR6: protected block, not included

SUBROUTINE_BLOCK 挡板电机手动控制:SBR7
TITLE=子程序注释
BEGIN
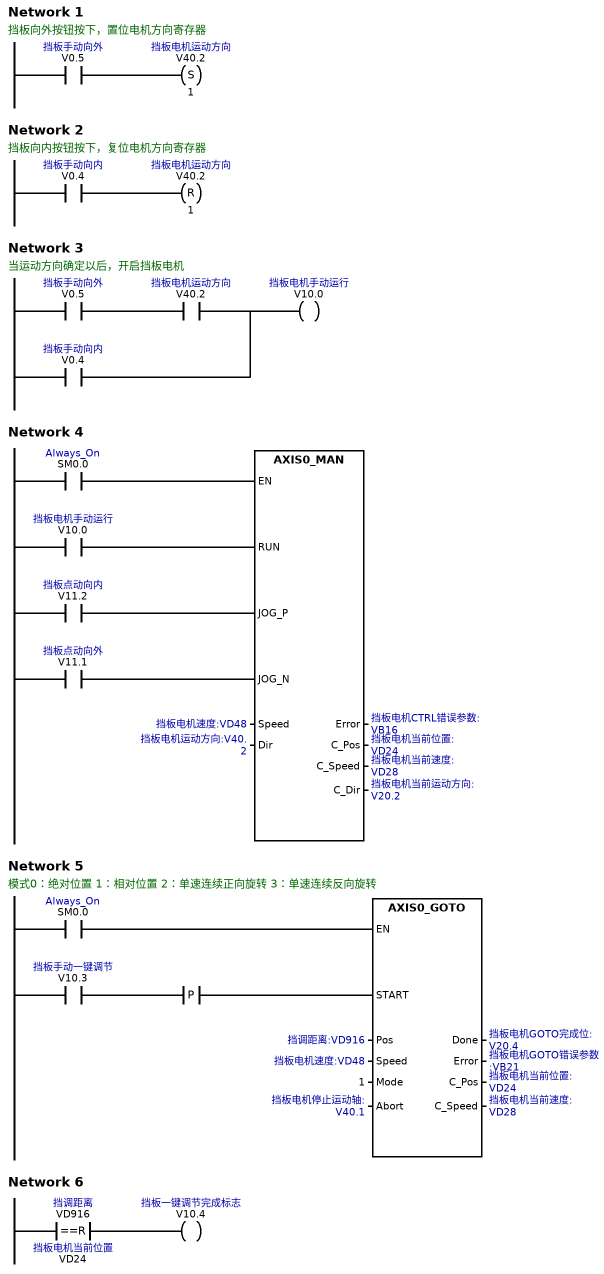
Network 1
// 挡板向外按钮按下，置位电机方向寄存器
LD     挡板手动向外:V0.5
S      挡板电机运动方向:V40.2, 1
Network 2
// 挡板向内按钮按下，复位电机方向寄存器
LD     挡板手动向内:V0.4
R      挡板电机运动方向:V40.2, 1
Network 3
// 当运动方向确定以后，开启挡板电机
LD     挡板手动向外:V0.5
A      挡板电机运动方向:V40.2
O      挡板手动向内:V0.4
=      挡板电机手动运行:V10.0
Network 4
LD     Always_On:SM0.0
=      L60.0
LD     挡板电机手动运行:V10.0
=      L63.7
LD     挡板点动向内:V11.2
=      L63.6
LD     挡板点动向外:V11.1
=      L63.5
LD     L60.0
CALL   AXIS0_MAN:SBR1, L63.7, L63.6, L63.5, 挡板电机速度:VD48, 挡板电机运动方向:V40.2, 挡板电机CTRL错误参数:VB16, 挡板电机当前位置:VD24, 挡板电机当前速度:VD28, 挡板电机当前运动方向:V20.2
Network 5
// 模式0：绝对位置 1：相对位置 2：单速连续正向旋转 3：单速连续反向旋转
LD     Always_On:SM0.0
=      L60.0
LD     挡板手动一键调节:V10.3
EU
=      L63.7
LD     L60.0
CALL   AXIS0_GOTO:SBR2, L63.7, 挡调距离:VD916, 挡板电机速度:VD48, 1, 挡板电机停止运动轴:V40.1, 挡板电机GOTO完成位:V20.4, 挡板电机GOTO错误参数:VB21, 挡板电机当前位置:VD24, 挡板电机当前速度:VD28
Network 6
LDR=   挡调距离:VD916, 挡板电机当前位置:VD24
=      挡板一键调节完成标志:V10.4
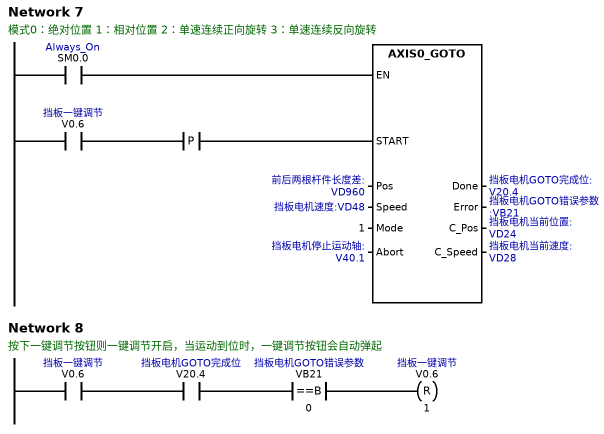
Network 7
// 模式0：绝对位置 1：相对位置 2：单速连续正向旋转 3：单速连续反向旋转
LD     Always_On:SM0.0
=      L60.0
LD     挡板一键调节:V0.6
EU
=      L63.7
LD     L60.0
CALL   AXIS0_GOTO:SBR2, L63.7, 前后两根杆件长度差:VD960, 挡板电机速度:VD48, 1, 挡板电机停止运动轴:V40.1, 挡板电机GOTO完成位:V20.4, 挡板电机GOTO错误参数:VB21, 挡板电机当前位置:VD24, 挡板电机当前速度:VD28
Network 8
// 按下一键调节按钮则一键调节开启，当运动到位时，一键调节按钮会自动弹起
LD     挡板一键调节:V0.6
A      挡板电机GOTO完成位:V20.4
AB=    挡板电机GOTO错误参数:VB21, 0
R      挡板一键调节:V0.6, 1
END_SUBROUTINE_BLOCK

// SBR8: protected block, not included

SUBROUTINE_BLOCK 下料电机手动控制:SBR9
TITLE=子程序注释
BEGIN
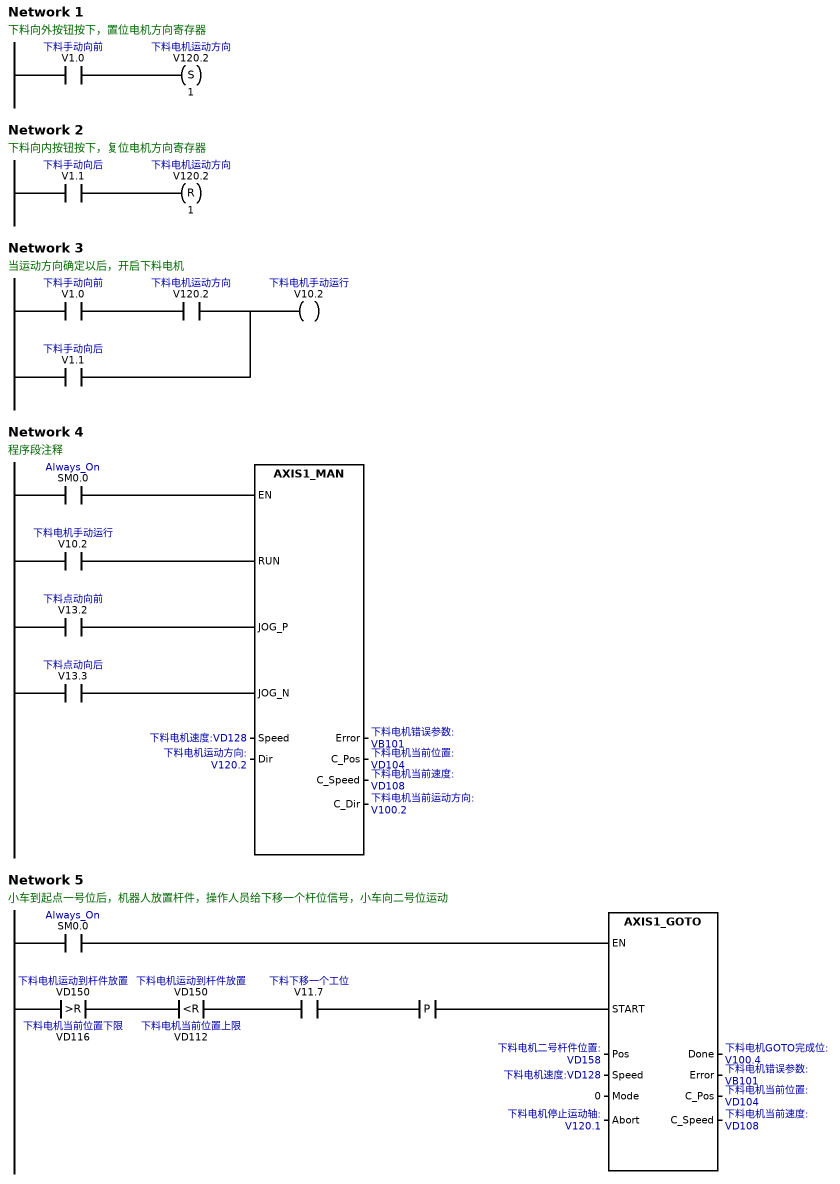
Network 1
// 下料向外按钮按下，置位电机方向寄存器
LD     下料手动向前:V1.0
S      下料电机运动方向:V120.2, 1
Network 2
// 下料向内按钮按下，复位电机方向寄存器
LD     下料手动向后:V1.1
R      下料电机运动方向:V120.2, 1
Network 3
// 当运动方向确定以后，开启下料电机
LD     下料手动向前:V1.0
A      下料电机运动方向:V120.2
O      下料手动向后:V1.1
=      下料电机手动运行:V10.2
Network 4
// 程序段注释
LD     Always_On:SM0.0
=      L60.0
LD     下料电机手动运行:V10.2
=      L63.7
LD     下料点动向前:V13.2
=      L63.6
LD     下料点动向后:V13.3
=      L63.5
LD     L60.0
CALL   AXIS1_MAN:SBR5, L63.7, L63.6, L63.5, 下料电机速度:VD128, 下料电机运动方向:V120.2, 下料电机错误参数:VB101, 下料电机当前位置:VD104, 下料电机当前速度:VD108, 下料电机当前运动方向:V100.2
Network 5
// 小车到起点一号位后，机器人放置杆件，操作人员给下移一个杆位信号，小车向二号位运动
LD     Always_On:SM0.0
=      L60.0
LDR>   下料电机运动到杆件放置:VD150, 下料电机当前位置下限:VD116
AR<    下料电机运动到杆件放置:VD150, 下料电机当前位置上限:VD112
A      下料下移一个工位:V11.7
EU
=      L63.7
LD     L60.0
CALL   AXIS1_GOTO:SBR6, L63.7, 下料电机二号杆件位置:VD158, 下料电机速度:VD128, 0, 下料电机停止运动轴:V120.1, 下料电机GOTO完成位:V100.4, 下料电机错误参数:VB101, 下料电机当前位置:VD104, 下料电机当前速度:VD108
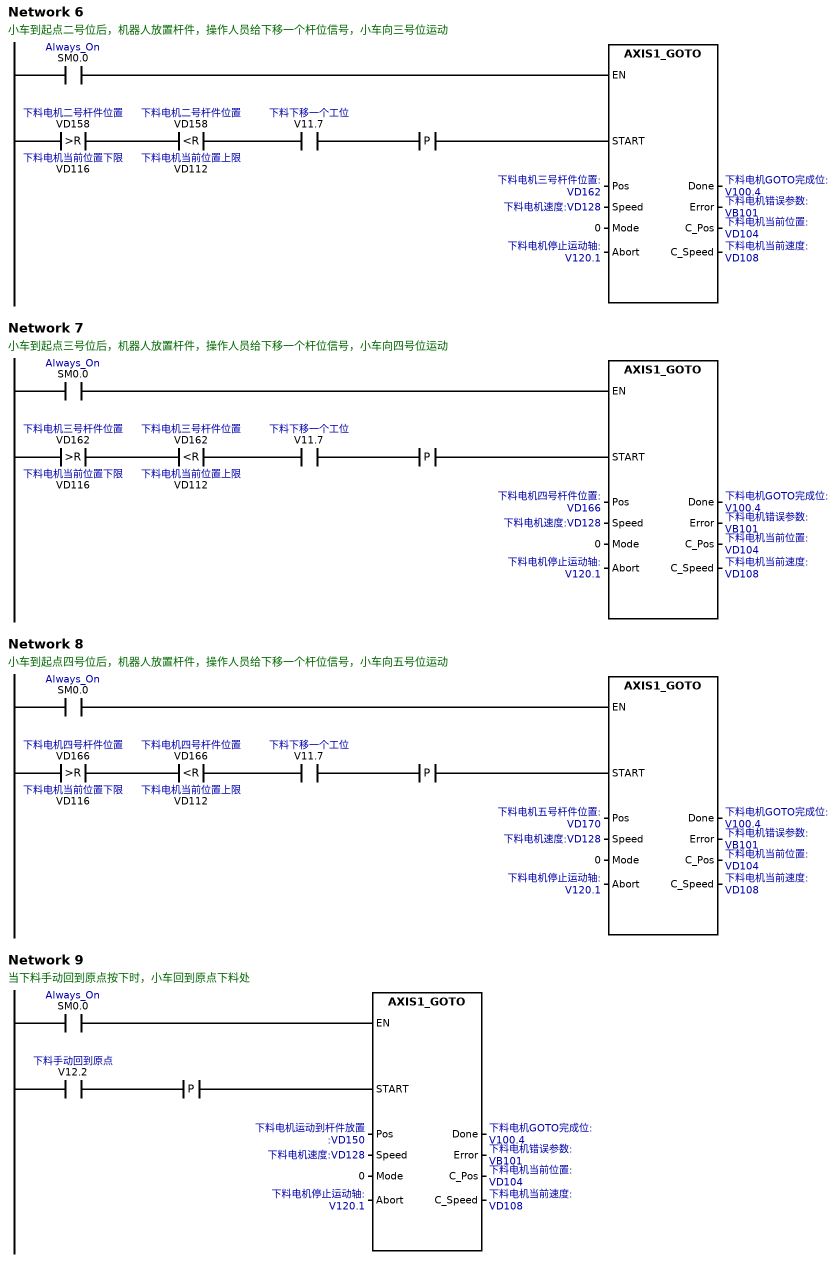
Network 6
// 小车到起点二号位后，机器人放置杆件，操作人员给下移一个杆位信号，小车向三号位运动
LD     Always_On:SM0.0
=      L60.0
LDR>   下料电机二号杆件位置:VD158, 下料电机当前位置下限:VD116
AR<    下料电机二号杆件位置:VD158, 下料电机当前位置上限:VD112
A      下料下移一个工位:V11.7
EU
=      L63.7
LD     L60.0
CALL   AXIS1_GOTO:SBR6, L63.7, 下料电机三号杆件位置:VD162, 下料电机速度:VD128, 0, 下料电机停止运动轴:V120.1, 下料电机GOTO完成位:V100.4, 下料电机错误参数:VB101, 下料电机当前位置:VD104, 下料电机当前速度:VD108
Network 7
// 小车到起点三号位后，机器人放置杆件，操作人员给下移一个杆位信号，小车向四号位运动
LD     Always_On:SM0.0
=      L60.0
LDR>   下料电机三号杆件位置:VD162, 下料电机当前位置下限:VD116
AR<    下料电机三号杆件位置:VD162, 下料电机当前位置上限:VD112
A      下料下移一个工位:V11.7
EU
=      L63.7
LD     L60.0
CALL   AXIS1_GOTO:SBR6, L63.7, 下料电机四号杆件位置:VD166, 下料电机速度:VD128, 0, 下料电机停止运动轴:V120.1, 下料电机GOTO完成位:V100.4, 下料电机错误参数:VB101, 下料电机当前位置:VD104, 下料电机当前速度:VD108
Network 8
// 小车到起点四号位后，机器人放置杆件，操作人员给下移一个杆位信号，小车向五号位运动
LD     Always_On:SM0.0
=      L60.0
LDR>   下料电机四号杆件位置:VD166, 下料电机当前位置下限:VD116
AR<    下料电机四号杆件位置:VD166, 下料电机当前位置上限:VD112
A      下料下移一个工位:V11.7
EU
=      L63.7
LD     L60.0
CALL   AXIS1_GOTO:SBR6, L63.7, 下料电机五号杆件位置:VD170, 下料电机速度:VD128, 0, 下料电机停止运动轴:V120.1, 下料电机GOTO完成位:V100.4, 下料电机错误参数:VB101, 下料电机当前位置:VD104, 下料电机当前速度:VD108
Network 9
// 当下料手动回到原点按下时，小车回到原点下料处
LD     Always_On:SM0.0
=      L60.0
LD     下料手动回到原点:V12.2
EU
=      L63.7
LD     L60.0
CALL   AXIS1_GOTO:SBR6, L63.7, 下料电机运动到杆件放置:VD150, 下料电机速度:VD128, 0, 下料电机停止运动轴:V120.1, 下料电机GOTO完成位:V100.4, 下料电机错误参数:VB101, 下料电机当前位置:VD104, 下料电机当前速度:VD108
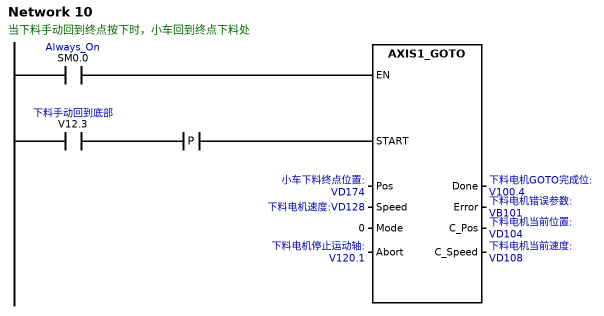
Network 10
// 当下料手动回到终点按下时，小车回到终点下料处
LD     Always_On:SM0.0
=      L60.0
LD     下料手动回到底部:V12.3
EU
=      L63.7
LD     L60.0
CALL   AXIS1_GOTO:SBR6, L63.7, 小车下料终点位置:VD174, 下料电机速度:VD128, 0, 下料电机停止运动轴:V120.1, 下料电机GOTO完成位:V100.4, 下料电机错误参数:VB101, 下料电机当前位置:VD104, 下料电机当前速度:VD108
END_SUBROUTINE_BLOCK

// SBR10: protected block, not included

// SBR11: protected block, not included

// SBR12: protected block, not included

// SBR13: protected block, not included

SUBROUTINE_BLOCK 上料初始化:SBR14
TITLE=子程序注释
BEGIN
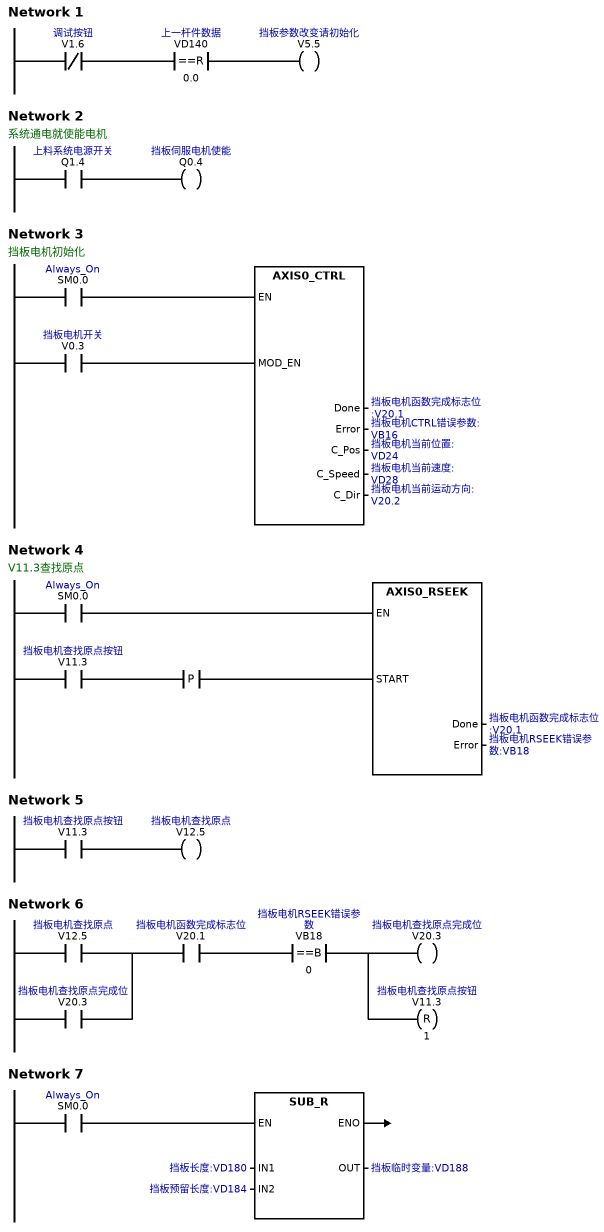
Network 1
LDN    调试按钮:V1.6
AR=    上一杆件数据:VD140, 0.0
=      挡板参数改变请初始化:V5.5
Network 2
// 系统通电就使能电机
LD     上料系统电源开关:Q1.4
=      挡板伺服电机使能:Q0.4
Network 3
// 挡板电机初始化
LD     Always_On:SM0.0
=      L60.0
LD     挡板电机开关:V0.3
=      L63.7
LD     L60.0
CALL   AXIS0_CTRL:SBR0, L63.7, 挡板电机函数完成标志位:V20.1, 挡板电机CTRL错误参数:VB16, 挡板电机当前位置:VD24, 挡板电机当前速度:VD28, 挡板电机当前运动方向:V20.2
Network 4
// V11.3查找原点
LD     Always_On:SM0.0
=      L60.0
LD     挡板电机查找原点按钮:V11.3
EU
=      L63.7
LD     L60.0
CALL   AXIS0_RSEEK:SBR3, L63.7, 挡板电机函数完成标志位:V20.1, 挡板电机RSEEK错误参数:VB18
Network 5
LD     挡板电机查找原点按钮:V11.3
=      挡板电机查找原点:V12.5
Network 6
LD     挡板电机查找原点:V12.5
O      挡板电机查找原点完成位:V20.3
A      挡板电机函数完成标志位:V20.1
AB=    挡板电机RSEEK错误参数:VB18, 0
=      挡板电机查找原点完成位:V20.3
R      挡板电机查找原点按钮:V11.3, 1
Network 7
LD     Always_On:SM0.0
MOVR   挡板长度:VD180, 挡板临时变量:VD188
-R     挡板预留长度:VD184, 挡板临时变量:VD188
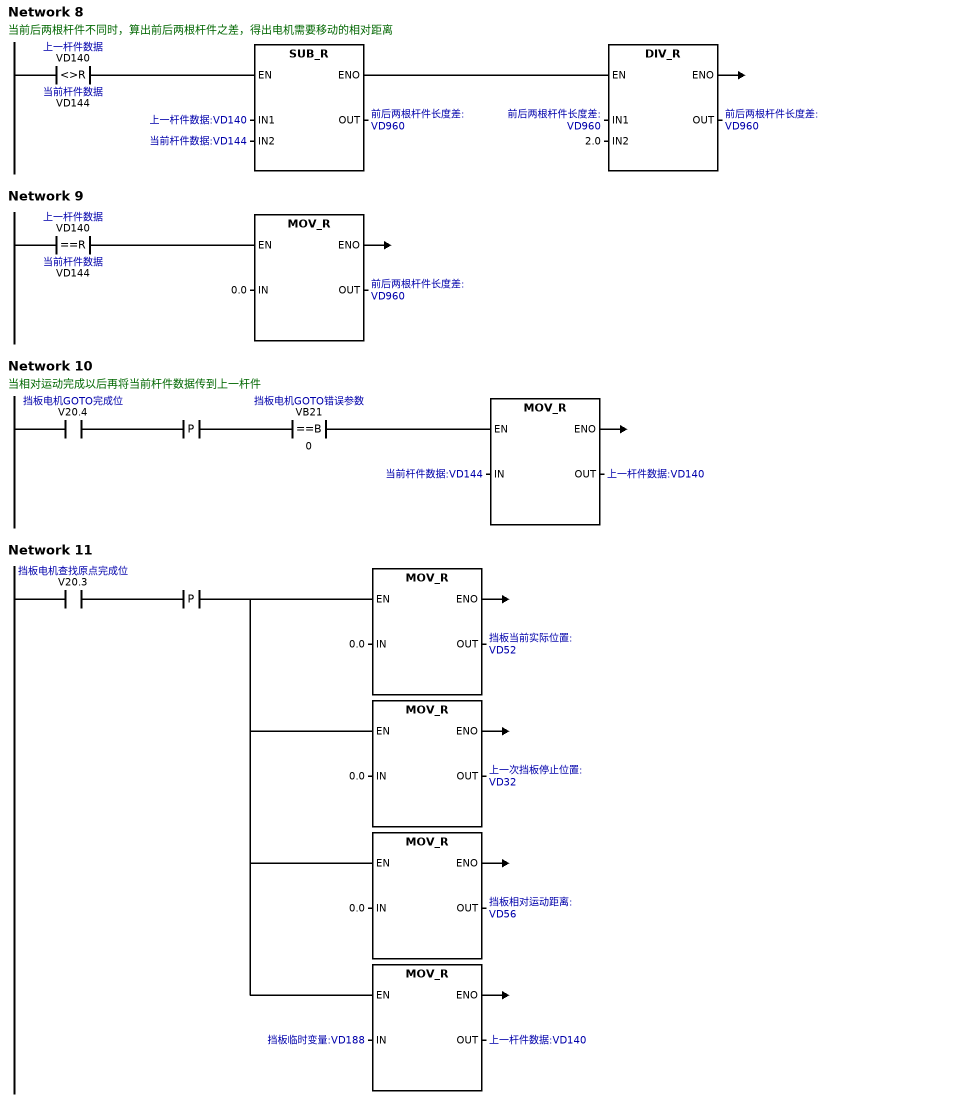
Network 8
// 当前后两根杆件不同时，算出前后两根杆件之差，得出电机需要移动的相对距离
LDR<>  上一杆件数据:VD140, 当前杆件数据:VD144
MOVR   上一杆件数据:VD140, 前后两根杆件长度差:VD960
AENO
-R     当前杆件数据:VD144, 前后两根杆件长度差:VD960
AENO
/R     2.0, 前后两根杆件长度差:VD960
Network 9
LDR=   上一杆件数据:VD140, 当前杆件数据:VD144
MOVR   0.0, 前后两根杆件长度差:VD960
Network 10
// 当相对运动完成以后再将当前杆件数据传到上一杆件
LD     挡板电机GOTO完成位:V20.4
EU
AB=    挡板电机GOTO错误参数:VB21, 0
MOVR   当前杆件数据:VD144, 上一杆件数据:VD140
Network 11
LD     挡板电机查找原点完成位:V20.3
EU
MOVR   0.0, 挡板当前实际位置:VD52
MOVR   0.0, 上一次挡板停止位置:VD32
MOVR   0.0, 挡板相对运动距离:VD56
MOVR   挡板临时变量:VD188, 上一杆件数据:VD140
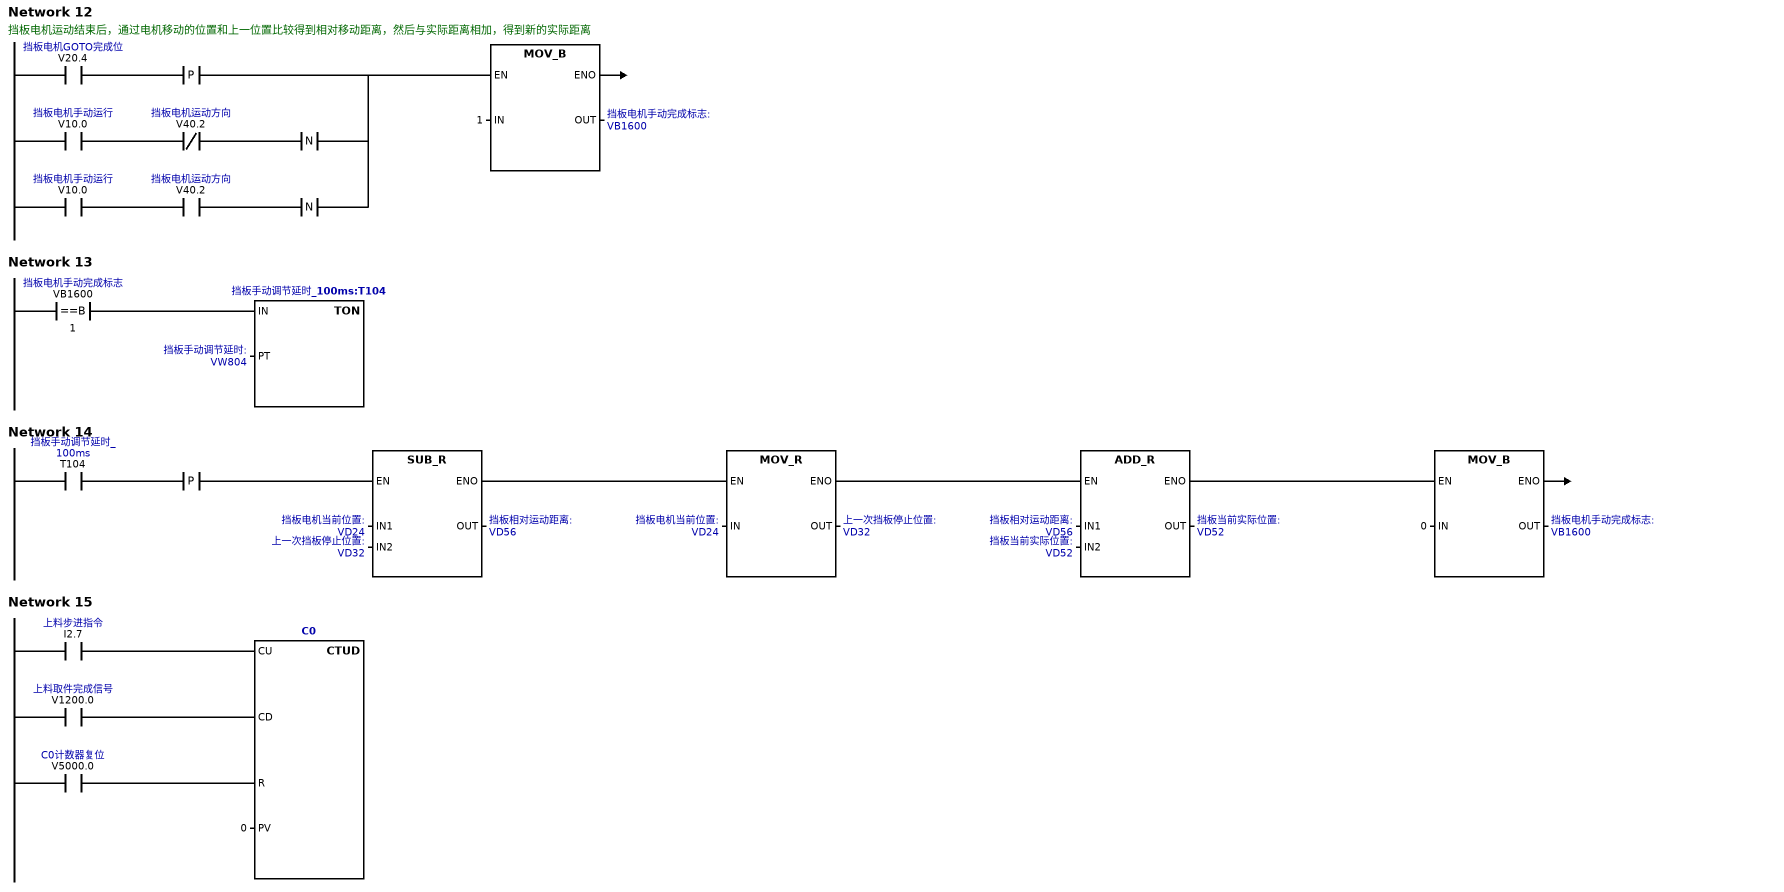
Network 12
// 挡板电机运动结束后，通过电机移动的位置和上一位置比较得到相对移动距离，然后与实际距离相加，得到新的实际距离
LD     挡板电机GOTO完成位:V20.4
EU
LD     挡板电机手动运行:V10.0
AN     挡板电机运动方向:V40.2
ED
OLD
LD     挡板电机手动运行:V10.0
A      挡板电机运动方向:V40.2
ED
OLD
MOVB   1, 挡板电机手动完成标志:VB1600
Network 13
LDB=   挡板电机手动完成标志:VB1600, 1
TON    挡板手动调节延时_100ms:T104, 挡板手动调节延时:VW804
Network 14
LD     挡板手动调节延时_100ms:T104
EU
MOVR   挡板电机当前位置:VD24, 挡板相对运动距离:VD56
AENO
-R     上一次挡板停止位置:VD32, 挡板相对运动距离:VD56
AENO
MOVR   挡板电机当前位置:VD24, 上一次挡板停止位置:VD32
AENO
+R     挡板相对运动距离:VD56, 挡板当前实际位置:VD52
AENO
MOVB   0, 挡板电机手动完成标志:VB1600
Network 15
LD     上料步进指令:I2.7
LD     上料取件完成信号:V1200.0
LD     C0计数器复位:V5000.0
CTUD   C0, 0
END_SUBROUTINE_BLOCK

SUBROUTINE_BLOCK 下料初始化:SBR15
TITLE=子程序注释
BEGIN
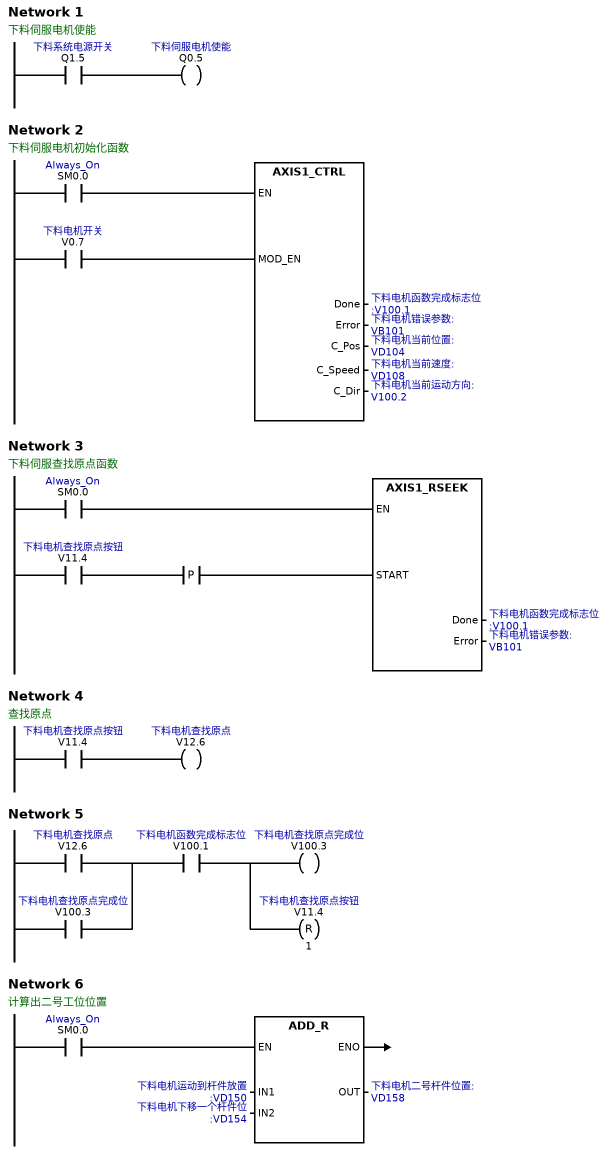
Network 1
// 下料伺服电机使能
LD     下料系统电源开关:Q1.5
=      下料伺服电机使能:Q0.5
Network 2
// 下料伺服电机初始化函数
LD     Always_On:SM0.0
=      L60.0
LD     下料电机开关:V0.7
=      L63.7
LD     L60.0
CALL   AXIS1_CTRL:SBR4, L63.7, 下料电机函数完成标志位:V100.1, 下料电机错误参数:VB101, 下料电机当前位置:VD104, 下料电机当前速度:VD108, 下料电机当前运动方向:V100.2
Network 3
// 下料伺服查找原点函数
LD     Always_On:SM0.0
=      L60.0
LD     下料电机查找原点按钮:V11.4
EU
=      L63.7
LD     L60.0
CALL   AXIS1_RSEEK:SBR8, L63.7, 下料电机函数完成标志位:V100.1, 下料电机错误参数:VB101
Network 4
// 查找原点
LD     下料电机查找原点按钮:V11.4
=      下料电机查找原点:V12.6
Network 5
LD     下料电机查找原点:V12.6
O      下料电机查找原点完成位:V100.3
A      下料电机函数完成标志位:V100.1
=      下料电机查找原点完成位:V100.3
R      下料电机查找原点按钮:V11.4, 1
Network 6
// 计算出二号工位位置
LD     Always_On:SM0.0
MOVR   下料电机运动到杆件放置:VD150, 下料电机二号杆件位置:VD158
+R     下料电机下移一个杆件位:VD154, 下料电机二号杆件位置:VD158
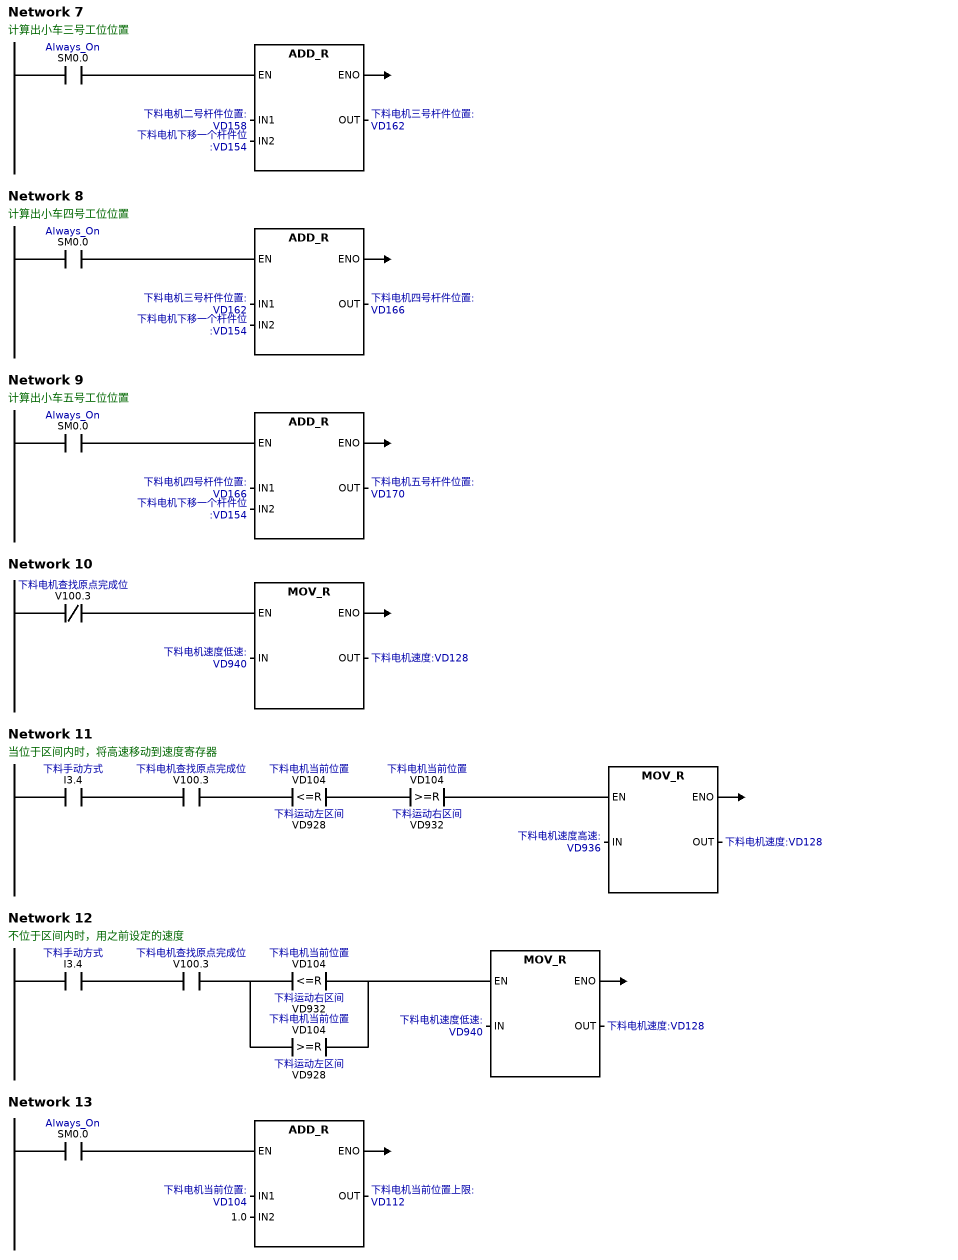
Network 7
// 计算出小车三号工位位置
LD     Always_On:SM0.0
MOVR   下料电机二号杆件位置:VD158, 下料电机三号杆件位置:VD162
+R     下料电机下移一个杆件位:VD154, 下料电机三号杆件位置:VD162
Network 8
// 计算出小车四号工位位置
LD     Always_On:SM0.0
MOVR   下料电机三号杆件位置:VD162, 下料电机四号杆件位置:VD166
+R     下料电机下移一个杆件位:VD154, 下料电机四号杆件位置:VD166
Network 9
// 计算出小车五号工位位置
LD     Always_On:SM0.0
MOVR   下料电机四号杆件位置:VD166, 下料电机五号杆件位置:VD170
+R     下料电机下移一个杆件位:VD154, 下料电机五号杆件位置:VD170
Network 10
LDN    下料电机查找原点完成位:V100.3
MOVR   下料电机速度低速:VD940, 下料电机速度:VD128
Network 11
// 当位于区间内时，将高速移动到速度寄存器
LD     下料手动方式:I3.4
A      下料电机查找原点完成位:V100.3
AR<=   下料电机当前位置:VD104, 下料运动左区间:VD928
AR>=   下料电机当前位置:VD104, 下料运动右区间:VD932
MOVR   下料电机速度高速:VD936, 下料电机速度:VD128
Network 12
// 不位于区间内时，用之前设定的速度
LD     下料手动方式:I3.4
A      下料电机查找原点完成位:V100.3
LDR<=  下料电机当前位置:VD104, 下料运动右区间:VD932
OR>=   下料电机当前位置:VD104, 下料运动左区间:VD928
ALD
MOVR   下料电机速度低速:VD940, 下料电机速度:VD128
Network 13
LD     Always_On:SM0.0
MOVR   下料电机当前位置:VD104, 下料电机当前位置上限:VD112
+R     1.0, 下料电机当前位置上限:VD112
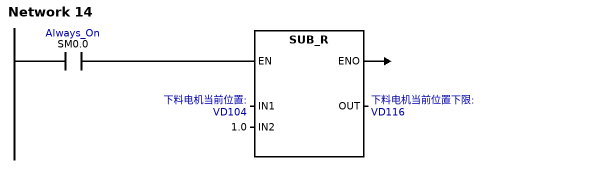
Network 14
LD     Always_On:SM0.0
MOVR   下料电机当前位置:VD104, 下料电机当前位置下限:VD116
-R     1.0, 下料电机当前位置下限:VD116
END_SUBROUTINE_BLOCK

SUBROUTINE_BLOCK 冷却初始化:SBR16
TITLE=子程序注释
BEGIN
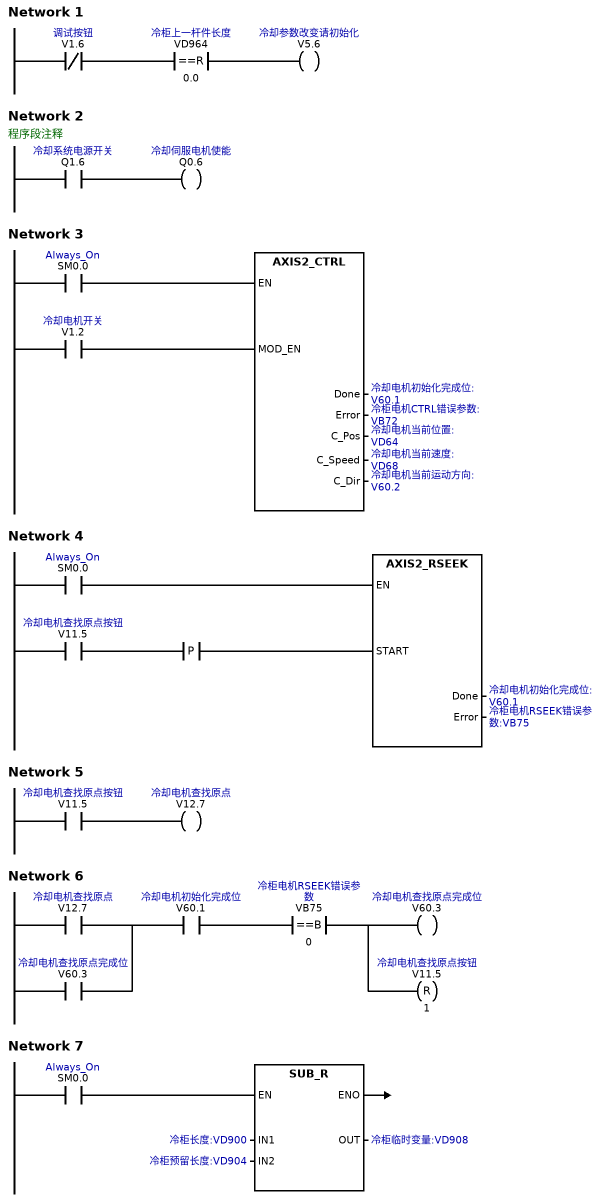
Network 1
LDN    调试按钮:V1.6
AR=    冷柜上一杆件长度:VD964, 0.0
=      冷却参数改变请初始化:V5.6
Network 2
// 程序段注释
LD     冷却系统电源开关:Q1.6
=      冷却伺服电机使能:Q0.6
Network 3
LD     Always_On:SM0.0
=      L60.0
LD     冷却电机开关:V1.2
=      L63.7
LD     L60.0
CALL   AXIS2_CTRL:SBR10, L63.7, 冷却电机初始化完成位:V60.1, 冷柜电机CTRL错误参数:VB72, 冷却电机当前位置:VD64, 冷却电机当前速度:VD68, 冷却电机当前运动方向:V60.2
Network 4
LD     Always_On:SM0.0
=      L60.0
LD     冷却电机查找原点按钮:V11.5
EU
=      L63.7
LD     L60.0
CALL   AXIS2_RSEEK:SBR13, L63.7, 冷却电机初始化完成位:V60.1, 冷柜电机RSEEK错误参数:VB75
Network 5
LD     冷却电机查找原点按钮:V11.5
=      冷却电机查找原点:V12.7
Network 6
LD     冷却电机查找原点:V12.7
O      冷却电机查找原点完成位:V60.3
A      冷却电机初始化完成位:V60.1
AB=    冷柜电机RSEEK错误参数:VB75, 0
=      冷却电机查找原点完成位:V60.3
R      冷却电机查找原点按钮:V11.5, 1
Network 7
LD     Always_On:SM0.0
MOVR   冷柜长度:VD900, 冷柜临时变量:VD908
-R     冷柜预留长度:VD904, 冷柜临时变量:VD908
